LIN {X 0,Y 573.244,Z 41.075,A -85,B 0,C 180,E1 -2290.525,E2 -2290.525} C_VEL
LIN {X 0,Y 573.235,Z 41.08,A -85,B 0,C 180,E1 -2293.359,E2 -2293.359} C_VEL
LIN {X 0,Y 573.243,Z 41.074,A -85,B 0,C 180,E1 -2296.331,E2 -2296.331} C_VEL
LIN {X 0,Y 573.273,Z 41.079,A -85,B 0,C 180,E1 -2299.477,E2 -2299.477} C_VEL
LIN {X 0,Y 573.234,Z 41.075,A -85,B 0,C 180,E1 -2302.192,E2 -2302.192} C_VEL
LIN {X 0,Y 573.268,Z 41.075,A -85,B 0,C 180,E1 -2304.816,E2 -2304.816} C_VEL
LIN {X 0,Y 573.253,Z 41.079,A -85,B 0,C 180,E1 -2307.355,E2 -2307.355} C_VEL
LIN {X 0,Y 573.245,Z 41.076,A -85,B 0,C 180,E1 -2310.511,E2 -2310.511} C_VEL
LIN {X 0,Y 573.249,Z 41.08,A -85,B 0,C 180,E1 -2313.024,E2 -2313.024} C_VEL
LIN {X 0,Y 573.273,Z 41.072,A -85,B 0,C 180,E1 -2315.366,E2 -2315.366} C_VEL
LIN {X 0,Y 573.228,Z 41.081,A -85,B 0,C 180,E1 -2318.419,E2 -2318.419} C_VEL
LIN {X 0,Y 573.276,Z 41.076,A -85,B 0,C 180,E1 -2320.728,E2 -2320.728} C_VEL
LIN {X 0,Y 573.25,Z 41.073,A -85,B 0,C 180,E1 -2323.622,E2 -2323.622} C_VEL
LIN {X 0,Y 573.271,Z 41.073,A -85,B 0,C 180,E1 -2325.807,E2 -2325.807} C_VEL
LIN {X 0,Y 573.261,Z 41.074,A -85,B 0,C 180,E1 -2328.745,E2 -2328.745} C_VEL
LIN {X 0,Y 573.288,Z 41.07,A -85,B 0,C 180,E1 -2331.541,E2 -2331.541} C_VEL
LIN {X 0,Y 573.285,Z 41.073,A -85,B 0,C 180,E1 -2334.372,E2 -2334.372} C_VEL
LIN {X 0,Y 573.305,Z 41.075,A -85,B 0,C 180,E1 -2337.893,E2 -2337.893} C_VEL
LIN {X 0,Y 573.327,Z 41.064,A -85,B 0,C 180,E1 -2340.703,E2 -2340.703} C_VEL
LIN {X 0,Y 573.233,Z 41.082,A -85,B 0,C 180,E1 -2343.515,E2 -2343.515} C_VEL
LIN {X 0,Y 573.285,Z 41.076,A -85,B 0,C 180,E1 -2345.628,E2 -2345.628} C_VEL
LIN {X 0,Y 573.264,Z 41.075,A -85,B 0,C 180,E1 -2347.75,E2 -2347.75} C_VEL
LIN {X 0,Y 573.262,Z 41.073,A -85,B 0,C 180,E1 -2350.597,E2 -2350.597} C_VEL
LIN {X 0,Y 573.261,Z 41.074,A -85,B 0,C 180,E1 -2352.749,E2 -2352.749} C_VEL
LIN {X 0,Y 573.233,Z 41.082,A -85,B 0,C 180,E1 -2354.92,E2 -2354.92} C_VEL
LIN {X 0,Y 573.237,Z 41.074,A -85,B 0,C 180,E1 -2357.849,E2 -2357.849} C_VEL
LIN {X 0,Y 573.24,Z 41.075,A -85,B 0,C 180,E1 -2360.077,E2 -2360.077} C_VEL
LIN {X 0,Y 573.23,Z 41.078,A -85,B 0,C 180,E1 -2362.338,E2 -2362.338} C_VEL
LIN {X 0,Y 573.244,Z 41.079,A -85,B 0,C 180,E1 -2364.382,E2 -2364.382} C_VEL
LIN {X 0,Y 572.614,Z 41.163,A -85,B 0,C 180,E1 -2364.968,E2 -2364.968} C_VEL
LIN {X 0,Y 569.754,Z 41.518,A -85,B 0,C 180,E1 -2365.919,E2 -2365.919} C_VEL
LIN {X 0,Y 567.309,Z 41.822,A -85,B 0,C 180,E1 -2366.685,E2 -2366.685} C_VEL
LIN {X 0,Y 566.253,Z 41.947,A -85,B 0,C 180,E1 -2367.276,E2 -2367.276} C_VEL
LIN {X 0,Y 566.165,Z 41.956,A -85,B 0,C 180,E1 -2367.476,E2 -2367.476} C_VEL
LIN {X 0,Y 566.198,Z 41.952,A -85,B 0,C 180,E1 -2369.769,E2 -2369.769} C_VEL
LIN {X 0,Y 566.202,Z 41.96,A -85,B 0,C 180,E1 -2372.43,E2 -2372.43} C_VEL
LIN {X 0,Y 566.168,Z 41.956,A -85,B 0,C 180,E1 -2374.988,E2 -2374.988} C_VEL
LIN {X 0,Y 566.191,Z 41.954,A -85,B 0,C 180,E1 -2377.462,E2 -2377.462} C_VEL
LIN {X 0,Y 566.206,Z 41.957,A -85,B 0,C 180,E1 -2380.2,E2 -2380.2} C_VEL
LIN {X 0,Y 566.178,Z 41.956,A -85,B 0,C 180,E1 -2383.057,E2 -2383.057} C_VEL
LIN {X 0,Y 566.159,Z 41.964,A -85,B 0,C 180,E1 -2386.054,E2 -2386.054} C_VEL
LIN {X 0,Y 566.158,Z 41.958,A -85,B 0,C 180,E1 -2388.859,E2 -2388.859} C_VEL
LIN {X 0,Y 566.201,Z 41.96,A -85,B 0,C 180,E1 -2391.444,E2 -2391.444} C_VEL
LIN {X 0,Y 566.144,Z 41.96,A -85,B 0,C 180,E1 -2394.307,E2 -2394.307} C_VEL
LIN {X 0,Y 566.194,Z 41.958,A -85,B 0,C 180,E1 -2396.896,E2 -2396.896} C_VEL
LIN {X 0,Y 566.213,Z 42.062,A -85,B 0,C 180,E1 -2398.293,E2 -2398.293} C_VEL
LIN {X 0,Y 566.339,Z 48.784,A -85,B 0,C 180,E1 -2399.623,E2 -2399.623} C_VEL
LIN {X 0,Y 566.243,Z 61.213,A -85,B 0,C 180,E1 -2402.061,E2 -2402.061} C_VEL
LIN {X 0,Y 567.205,Z 67.215,A -85,B 0,C 180,E1 -2402.163,E2 -2402.163} C_VEL
LIN {X 0,Y 566.982,Z 167.233,A -85,B 0,C 180,E1 -2403.452,E2 -2403.452} C_VEL
LIN {X 0,Y 566.828,Z 180.305,A -85,B 0,C 180,E1 -2403.763,E2 -2403.763} C_VEL
LIN {X 0,Y 566.757,Z 193.318,A -85,B 0,C 180,E1 -2404.229,E2 -2404.229} C_VEL
LIN {X 0,Y 566.573,Z 205.2,A -85,B 0,C 180,E1 -2404.81,E2 -2404.81} C_VEL
LIN {X 0,Y 566.359,Z 216.706,A -85,B 0,C 180,E1 -2405.534,E2 -2405.534} C_VEL
LIN {X 0,Y 566.298,Z 227.724,A -85,B 0,C 180,E1 -2406.407,E2 -2406.407} C_VEL
LIN {X 0,Y 566.15,Z 237.413,A -85,B 0,C 180,E1 -2407.368,E2 -2407.368} C_VEL
LIN {X 0,Y 566.067,Z 245.994,A -85,B 0,C 180,E1 -2408.416,E2 -2408.416} C_VEL
LIN {X 0,Y 566.006,Z 252.944,A -85,B 0,C 180,E1 -2409.466,E2 -2409.466} C_VEL
LIN {X 0,Y 565.942,Z 259.355,A -85,B 0,C 180,E1 -2410.699,E2 -2410.699} C_VEL
LIN {X 0,Y 565.913,Z 264.167,A -85,B 0,C 180,E1 -2411.913,E2 -2411.913} C_VEL
LIN {X 0,Y 565.862,Z 267.344,A -85,B 0,C 180,E1 -2413.008,E2 -2413.008} C_VEL
LIN {X 0,Y 565.813,Z 269.563,A -85,B 0,C 180,E1 -2414.142,E2 -2414.142} C_VEL
LIN {X 0,Y 565.807,Z 270.469,A -85,B 0,C 180,E1 -2414.88,E2 -2414.88} C_VEL
LIN {X 0,Y 565.855,Z 270.917,A -85,B 0,C 180,E1 -2415.645,E2 -2415.645} C_VEL
LIN {X 0,Y 565.866,Z 270.938,A -85,B 0,C 180,E1 -2416.351,E2 -2416.351} C_VEL
LIN {X 0,Y 565.845,Z 270.566,A -85,B 0,C 180,E1 -2417.082,E2 -2417.082} C_VEL
LIN {X 0,Y 565.867,Z 269.774,A -85,B 0,C 180,E1 -2417.811,E2 -2417.811} C_VEL
LIN {X 0,Y 565.908,Z 267.91,A -85,B 0,C 180,E1 -2418.845,E2 -2418.845} C_VEL
LIN {X 0,Y 565.925,Z 264.812,A -85,B 0,C 180,E1 -2419.988,E2 -2419.988} C_VEL
LIN {X 0,Y 565.944,Z 260.793,A -85,B 0,C 180,E1 -2421.07,E2 -2421.07} C_VEL
LIN {X 0,Y 565.986,Z 254.613,A -85,B 0,C 180,E1 -2422.329,E2 -2422.329} C_VEL
LIN {X 0,Y 566.023,Z 248.098,A -85,B 0,C 180,E1 -2423.377,E2 -2423.377} C_VEL
LIN {X 0,Y 566.099,Z 239.606,A -85,B 0,C 180,E1 -2424.479,E2 -2424.479} C_VEL
LIN {X 0,Y 566.237,Z 231.088,A -85,B 0,C 180,E1 -2425.373,E2 -2425.373} C_VEL
LIN {X 0,Y 566.385,Z 220.63,A -85,B 0,C 180,E1 -2426.265,E2 -2426.265} C_VEL
LIN {X 0,Y 566.535,Z 210.305,A -85,B 0,C 180,E1 -2426.978,E2 -2426.978} C_VEL
LIN {X 0,Y 566.7,Z 199.046,A -85,B 0,C 180,E1 -2427.601,E2 -2427.601} C_VEL
LIN {X 0,Y 566.746,Z 187.532,A -85,B 0,C 180,E1 -2428.09,E2 -2428.09} C_VEL
LIN {X 0,Y 566.884,Z 175.12,A -85,B 0,C 180,E1 -2428.468,E2 -2428.468} C_VEL
LIN {X 0,Y 566.961,Z 162.555,A -85,B 0,C 180,E1 -2428.713,E2 -2428.713} C_VEL
LIN {X 0,Y 567.066,Z 66.094,A -85,B 0,C 180,E1 -2429.945,E2 -2429.945} C_VEL
LIN {X 0,Y 566.19,Z 61.097,A -85,B 0,C 180,E1 -2430.045,E2 -2430.045} C_VEL
LIN {X 0,Y 566.414,Z 46.902,A -85,B 0,C 180,E1 -2432.845,E2 -2432.845} C_VEL
LIN {X 0,Y 566.211,Z 41.956,A -85,B 0,C 180,E1 -2433.826,E2 -2433.826} C_VEL
LIN {X 0,Y 566.26,Z 41.946,A -85,B 0,C 180,E1 -2435.699,E2 -2435.699} C_VEL
LIN {X 0,Y 566.232,Z 41.957,A -85,B 0,C 180,E1 -2438.566,E2 -2438.566} C_VEL
LIN {X 0,Y 566.249,Z 41.945,A -85,B 0,C 180,E1 -2441.454,E2 -2441.454} C_VEL
LIN {X 0,Y 566.241,Z 41.955,A -85,B 0,C 180,E1 -2444.506,E2 -2444.506} C_VEL
LIN {X 0,Y 566.204,Z 41.951,A -85,B 0,C 180,E1 -2447.332,E2 -2447.332} C_VEL
LIN {X 0,Y 566.212,Z 41.958,A -85,B 0,C 180,E1 -2450.337,E2 -2450.337} C_VEL
LIN {X 0,Y 566.175,Z 41.955,A -85,B 0,C 180,E1 -2453.281,E2 -2453.281} C_VEL
LIN {X 0,Y 566.215,Z 41.954,A -85,B 0,C 180,E1 -2455.749,E2 -2455.749} C_VEL
LIN {X 0,Y 566.209,Z 41.956,A -85,B 0,C 180,E1 -2458.202,E2 -2458.202} C_VEL
LIN {X 0,Y 566.195,Z 41.952,A -85,B 0,C 180,E1 -2461.076,E2 -2461.076} C_VEL
LIN {X 0,Y 566.218,Z 41.958,A -85,B 0,C 180,E1 -2463.734,E2 -2463.734} C_VEL
LIN {X 0,Y 566.212,Z 41.95,A -85,B 0,C 180,E1 -2466.569,E2 -2466.569} C_VEL
LIN {X 0,Y 566.218,Z 41.957,A -85,B 0,C 180,E1 -2469.685,E2 -2469.685} C_VEL
LIN {X 0,Y 566.205,Z 41.953,A -85,B 0,C 180,E1 -2472.917,E2 -2472.917} C_VEL
LIN {X 0,Y 566.198,Z 41.952,A -85,B 0,C 180,E1 -2476.049,E2 -2476.049} C_VEL
LIN {X 0,Y 566.207,Z 41.96,A -85,B 0,C 180,E1 -2479.214,E2 -2479.214} C_VEL
LIN {X 0,Y 566.19,Z 41.955,A -85,B 0,C 180,E1 -2481.637,E2 -2481.637} C_VEL
LIN {X 0,Y 566.167,Z 41.956,A -85,B 0,C 180,E1 -2484.308,E2 -2484.308} C_VEL
LIN {X 0,Y 566.223,Z 41.957,A -85,B 0,C 180,E1 -2486.898,E2 -2486.898} C_VEL
LIN {X 0,Y 566.184,Z 41.955,A -85,B 0,C 180,E1 -2489.407,E2 -2489.407} C_VEL
LIN {X 0,Y 566.215,Z 41.949,A -85,B 0,C 180,E1 -2491.857,E2 -2491.857} C_VEL
LIN {X 0,Y 566.213,Z 41.953,A -85,B 0,C 180,E1 -2494.251,E2 -2494.251} C_VEL
LIN {X 0,Y 566.176,Z 41.962,A -85,B 0,C 180,E1 -2496.718,E2 -2496.718} C_VEL
LIN {X 0,Y 566.215,Z 41.95,A -85,B 0,C 180,E1 -2499.663,E2 -2499.663} C_VEL
LIN {X 0,Y 566.201,Z 41.956,A -85,B 0,C 180,E1 -2502.668,E2 -2502.668} C_VEL
LIN {X 0,Y 566.237,Z 41.948,A -85,B 0,C 180,E1 -2505.627,E2 -2505.627} C_VEL
LIN {X 0,Y 566.238,Z 41.949,A -85,B 0,C 180,E1 -2508.675,E2 -2508.675} C_VEL
LIN {X 0,Y 566.23,Z 41.949,A -85,B 0,C 180,E1 -2511.434,E2 -2511.434} C_VEL
LIN {X 0,Y 566.256,Z 41.949,A -85,B 0,C 180,E1 -2514.301,E2 -2514.301} C_VEL
LIN {X 0,Y 566.28,Z 41.951,A -85,B 0,C 180,E1 -2517.866,E2 -2517.866} C_VEL
LIN {X 0,Y 566.301,Z 41.939,A -85,B 0,C 180,E1 -2520.711,E2 -2520.711} C_VEL
LIN {X 0,Y 566.27,Z 41.943,A -85,B 0,C 180,E1 -2522.845,E2 -2522.845} C_VEL
LIN {X 0,Y 566.255,Z 41.952,A -85,B 0,C 180,E1 -2525.698,E2 -2525.698} C_VEL
LIN {X 0,Y 566.207,Z 41.95,A -85,B 0,C 180,E1 -2528.566,E2 -2528.566} C_VEL
LIN {X 0,Y 566.244,Z 41.954,A -85,B 0,C 180,E1 -2531.454,E2 -2531.454} C_VEL
LIN {X 0,Y 566.232,Z 41.948,A -85,B 0,C 180,E1 -2534.505,E2 -2534.505} C_VEL
LIN {X 0,Y 566.2,Z 41.958,A -85,B 0,C 180,E1 -2537.332,E2 -2537.332} C_VEL
LIN {X 0,Y 566.209,Z 41.951,A -85,B 0,C 180,E1 -2540.337,E2 -2540.337} C_VEL
LIN {X 0,Y 566.17,Z 41.96,A -85,B 0,C 180,E1 -2543.281,E2 -2543.281} C_VEL
LIN {X 0,Y 566.208,Z 41.95,A -85,B 0,C 180,E1 -2545.749,E2 -2545.749} C_VEL
LIN {X 0,Y 566.205,Z 41.952,A -85,B 0,C 180,E1 -2548.202,E2 -2548.202} C_VEL
LIN {X 0,Y 566.192,Z 41.956,A -85,B 0,C 180,E1 -2551.076,E2 -2551.076} C_VEL
LIN {X 0,Y 566.213,Z 41.95,A -85,B 0,C 180,E1 -2553.734,E2 -2553.734} C_VEL
LIN {X 0,Y 566.202,Z 41.96,A -85,B 0,C 180,E1 -2556.57,E2 -2556.57} C_VEL
LIN {X 0,Y 566.217,Z 41.95,A -85,B 0,C 180,E1 -2559.686,E2 -2559.686} C_VEL
LIN {X 0,Y 566.203,Z 41.952,A -85,B 0,C 180,E1 -2562.917,E2 -2562.917} C_VEL
LIN {X 0,Y 566.196,Z 41.96,A -85,B 0,C 180,E1 -2566.049,E2 -2566.049} C_VEL
LIN {X 0,Y 566.206,Z 41.951,A -85,B 0,C 180,E1 -2569.215,E2 -2569.215} C_VEL
LIN {X 0,Y 566.184,Z 41.958,A -85,B 0,C 180,E1 -2571.636,E2 -2571.636} C_VEL
LIN {X 0,Y 566.165,Z 41.959,A -85,B 0,C 180,E1 -2574.308,E2 -2574.308} C_VEL
LIN {X 0,Y 566.208,Z 41.95,A -85,B 0,C 180,E1 -2576.897,E2 -2576.897} C_VEL
LIN {X 0,Y 566.177,Z 41.959,A -85,B 0,C 180,E1 -2579.407,E2 -2579.407} C_VEL
LIN {X 0,Y 566.215,Z 41.957,A -85,B 0,C 180,E1 -2581.857,E2 -2581.857} C_VEL
LIN {X 0,Y 566.21,Z 41.954,A -85,B 0,C 180,E1 -2584.251,E2 -2584.251} C_VEL
LIN {X 0,Y 566.261,Z 42.133,A -85,B 0,C 180,E1 -2585.676,E2 -2585.676} C_VEL
LIN {X 0,Y 567.069,Z 47.897,A -85,B 0,C 180,E1 -2586.509,E2 -2586.509} C_VEL
LIN {X 0,Y 566.843,Z 66.898,A -85,B 0,C 180,E1 -2589.117,E2 -2589.117} C_VEL
LIN {X 0,Y 566.688,Z 87.811,A -85,B 0,C 180,E1 -2591.938,E2 -2591.938} C_VEL
LIN {X 0,Y 566.434,Z 110.038,A -85,B 0,C 180,E1 -2594.897,E2 -2594.897} C_VEL
LIN {X 0,Y 566.431,Z 118.271,A -85,B 0,C 180,E1 -2595.987,E2 -2595.987} C_VEL
LIN {X 0,Y 567.159,Z 125.154,A -85,B 0,C 180,E1 -2596.095,E2 -2596.095} C_VEL
LIN {X 0,Y 566.941,Z 226.934,A -85,B 0,C 180,E1 -2597.402,E2 -2597.402} C_VEL
LIN {X 0,Y 566.859,Z 240.209,A -85,B 0,C 180,E1 -2597.719,E2 -2597.719} C_VEL
LIN {X 0,Y 566.76,Z 252.371,A -85,B 0,C 180,E1 -2598.148,E2 -2598.148} C_VEL
LIN {X 0,Y 566.604,Z 264.234,A -85,B 0,C 180,E1 -2598.712,E2 -2598.712} C_VEL
LIN {X 0,Y 566.442,Z 276.19,A -85,B 0,C 180,E1 -2599.455,E2 -2599.455} C_VEL
LIN {X 0,Y 566.325,Z 286.603,A -85,B 0,C 180,E1 -2600.265,E2 -2600.265} C_VEL
LIN {X 0,Y 566.207,Z 295.111,A -85,B 0,C 180,E1 -2601.074,E2 -2601.074} C_VEL
LIN {X 0,Y 566.112,Z 302.959,A -85,B 0,C 180,E1 -2601.971,E2 -2601.971} C_VEL
LIN {X 0,Y 566.004,Z 310.621,A -85,B 0,C 180,E1 -2603.046,E2 -2603.046} C_VEL
LIN {X 0,Y 566.004,Z 317.678,A -85,B 0,C 180,E1 -2604.299,E2 -2604.299} C_VEL
LIN {X 0,Y 565.933,Z 322.372,A -85,B 0,C 180,E1 -2605.37,E2 -2605.37} C_VEL
LIN {X 0,Y 565.927,Z 325.958,A -85,B 0,C 180,E1 -2606.44,E2 -2606.44} C_VEL
LIN {X 0,Y 565.878,Z 327.807,A -85,B 0,C 180,E1 -2607.152,E2 -2607.152} C_VEL
LIN {X 0,Y 565.846,Z 330.183,A -85,B 0,C 180,E1 -2608.576,E2 -2608.576} C_VEL
LIN {X 0,Y 565.839,Z 331,A -85,B 0,C 180,E1 -2610,E2 -2610} C_VEL
LIN {X 0,Y 565.846,Z 330.185,A -85,B 0,C 180,E1 -2611.423,E2 -2611.423} C_VEL
LIN {X 0,Y 565.878,Z 327.811,A -85,B 0,C 180,E1 -2612.847,E2 -2612.847} C_VEL
LIN {X 0,Y 565.926,Z 324.896,A -85,B 0,C 180,E1 -2613.916,E2 -2613.916} C_VEL
LIN {X 0,Y 565.878,Z 320.949,A -85,B 0,C 180,E1 -2614.987,E2 -2614.987} C_VEL
LIN {X 0,Y 566.004,Z 315.869,A -85,B 0,C 180,E1 -2616.058,E2 -2616.058} C_VEL
LIN {X 0,Y 566.04,Z 309.469,A -85,B 0,C 180,E1 -2617.132,E2 -2617.132} C_VEL
LIN {X 0,Y 566.133,Z 301.48,A -85,B 0,C 180,E1 -2618.207,E2 -2618.207} C_VEL
LIN {X 0,Y 566.228,Z 293.336,A -85,B 0,C 180,E1 -2619.105,E2 -2619.105} C_VEL
LIN {X 0,Y 566.342,Z 283.401,A -85,B 0,C 180,E1 -2620.005,E2 -2620.005} C_VEL
LIN {X 0,Y 566.514,Z 272.293,A -85,B 0,C 180,E1 -2620.807,E2 -2620.807} C_VEL
LIN {X 0,Y 566.612,Z 261.177,A -85,B 0,C 180,E1 -2621.446,E2 -2621.446} C_VEL
LIN {X 0,Y 566.738,Z 248.984,A -85,B 0,C 180,E1 -2621.988,E2 -2621.988} C_VEL
LIN {X 0,Y 566.886,Z 236.185,A -85,B 0,C 180,E1 -2622.394,E2 -2622.394} C_VEL
LIN {X 0,Y 566.99,Z 224.122,A -85,B 0,C 180,E1 -2622.641,E2 -2622.641} C_VEL
LIN {X 0,Y 567.069,Z 122.874,A -85,B 0,C 180,E1 -2623.937,E2 -2623.937} C_VEL
LIN {X 0,Y 566.429,Z 118.184,A -85,B 0,C 180,E1 -2624.024,E2 -2624.024} C_VEL
LIN {X 0,Y 566.582,Z 96.456,A -85,B 0,C 180,E1 -2626.903,E2 -2626.903} C_VEL
LIN {X 0,Y 566.79,Z 75.205,A -85,B 0,C 180,E1 -2629.748,E2 -2629.748} C_VEL
LIN {X 0,Y 566.963,Z 54.272,A -85,B 0,C 180,E1 -2632.598,E2 -2632.598} C_VEL
LIN {X 0,Y 566.957,Z 45.828,A -85,B 0,C 180,E1 -2633.766,E2 -2633.766} C_VEL
LIN {X 0,Y 566.256,Z 41.954,A -85,B 0,C 180,E1 -2634.348,E2 -2634.348} C_VEL
LIN {X 0,Y 566.213,Z 41.952,A -85,B 0,C 180,E1 -2637.339,E2 -2637.339} C_VEL
LIN {X 0,Y 566.201,Z 41.955,A -85,B 0,C 180,E1 -2639.768,E2 -2639.768} C_VEL
LIN {X 0,Y 566.204,Z 41.957,A -85,B 0,C 180,E1 -2642.429,E2 -2642.429} C_VEL
LIN {X 0,Y 566.212,Z 41.95,A -85,B 0,C 180,E1 -2644.994,E2 -2644.994} C_VEL
LIN {X 0,Y 566.197,Z 41.955,A -85,B 0,C 180,E1 -2647.46,E2 -2647.46} C_VEL
LIN {X 0,Y 566.206,Z 41.955,A -85,B 0,C 180,E1 -2650.199,E2 -2650.199} C_VEL
LIN {X 0,Y 566.199,Z 41.953,A -85,B 0,C 180,E1 -2653.054,E2 -2653.054} C_VEL
LIN {X 0,Y 566.197,Z 41.954,A -85,B 0,C 180,E1 -2656.048,E2 -2656.048} C_VEL
LIN {X 0,Y 566.207,Z 41.952,A -85,B 0,C 180,E1 -2658.863,E2 -2658.863} C_VEL
LIN {X 0,Y 566.188,Z 41.957,A -85,B 0,C 180,E1 -2661.637,E2 -2661.637} C_VEL
LIN {X 0,Y 566.212,Z 41.95,A -85,B 0,C 180,E1 -2664.311,E2 -2664.311} C_VEL
LIN {X 0,Y 566.227,Z 41.954,A -85,B 0,C 180,E1 -2666.898,E2 -2666.898} C_VEL
LIN {X 0,Y 566.183,Z 41.957,A -85,B 0,C 180,E1 -2669.407,E2 -2669.407} C_VEL
LIN {X 0,Y 566.227,Z 41.948,A -85,B 0,C 180,E1 -2671.858,E2 -2671.858} C_VEL
LIN {X 0,Y 566.212,Z 41.951,A -85,B 0,C 180,E1 -2674.251,E2 -2674.251} C_VEL
LIN {X 0,Y 566.189,Z 41.961,A -85,B 0,C 180,E1 -2676.714,E2 -2676.714} C_VEL
LIN {X 0,Y 566.212,Z 41.95,A -85,B 0,C 180,E1 -2679.663,E2 -2679.663} C_VEL
LIN {X 0,Y 566.198,Z 41.958,A -85,B 0,C 180,E1 -2682.668,E2 -2682.668} C_VEL
LIN {X 0,Y 566.232,Z 41.948,A -85,B 0,C 180,E1 -2685.627,E2 -2685.627} C_VEL
LIN {X 0,Y 566.233,Z 41.95,A -85,B 0,C 180,E1 -2688.675,E2 -2688.675} C_VEL
LIN {X 0,Y 566.232,Z 41.948,A -85,B 0,C 180,E1 -2691.434,E2 -2691.434} C_VEL
LIN {X 0,Y 566.254,Z 41.95,A -85,B 0,C 180,E1 -2694.302,E2 -2694.302} C_VEL
LIN {X 0,Y 566.276,Z 41.95,A -85,B 0,C 180,E1 -2697.866,E2 -2697.866} C_VEL
LIN {X 0,Y 566.298,Z 41.939,A -85,B 0,C 180,E1 -2700.711,E2 -2700.711} C_VEL
LIN {X 0,Y 566.268,Z 41.942,A -85,B 0,C 180,E1 -2702.846,E2 -2702.846} C_VEL
LIN {X 0,Y 566.252,Z 41.951,A -85,B 0,C 180,E1 -2705.699,E2 -2705.699} C_VEL
LIN {X 0,Y 566.199,Z 41.951,A -85,B 0,C 180,E1 -2708.566,E2 -2708.566} C_VEL
LIN {X 0,Y 566.24,Z 41.952,A -85,B 0,C 180,E1 -2711.455,E2 -2711.455} C_VEL
LIN {X 0,Y 566.227,Z 41.949,A -85,B 0,C 180,E1 -2714.505,E2 -2714.505} C_VEL
LIN {X 0,Y 566.196,Z 41.956,A -85,B 0,C 180,E1 -2717.332,E2 -2717.332} C_VEL
LIN {X 0,Y 566.206,Z 41.953,A -85,B 0,C 180,E1 -2720.338,E2 -2720.338} C_VEL
LIN {X 0,Y 566.167,Z 41.958,A -85,B 0,C 180,E1 -2723.281,E2 -2723.281} C_VEL
LIN {X 0,Y 566.203,Z 41.95,A -85,B 0,C 180,E1 -2725.75,E2 -2725.75} C_VEL
LIN {X 0,Y 566.165,Z 41.956,A -85,B 0,C 180,E1 -2727.476,E2 -2727.476} C_VEL
LIN {X 0,Y 565.495,Z 42.044,A -85,B 0,C 180,E1 -2728.07,E2 -2728.07} C_VEL
LIN {X 0,Y 562.644,Z 42.396,A -85,B 0,C 180,E1 -2729.034,E2 -2729.034} C_VEL
LIN {X 0,Y 560.242,Z 42.696,A -85,B 0,C 180,E1 -2729.81,E2 -2729.81} C_VEL
LIN {X 0,Y 559.217,Z 42.83,A -85,B 0,C 180,E1 -2730.409,E2 -2730.409} C_VEL
LIN {X 0,Y 559.136,Z 42.833,A -85,B 0,C 180,E1 -2730.612,E2 -2730.612} C_VEL
LIN {X 0,Y 559.152,Z 42.834,A -85,B 0,C 180,E1 -2732.716,E2 -2732.716} C_VEL
LIN {X 0,Y 559.117,Z 42.833,A -85,B 0,C 180,E1 -2735.325,E2 -2735.325} C_VEL
LIN {X 0,Y 559.129,Z 42.841,A -85,B 0,C 180,E1 -2738.018,E2 -2738.018} C_VEL
LIN {X 0,Y 559.152,Z 42.829,A -85,B 0,C 180,E1 -2740.813,E2 -2740.813} C_VEL
LIN {X 0,Y 559.107,Z 42.844,A -85,B 0,C 180,E1 -2743.738,E2 -2743.738} C_VEL
LIN {X 0,Y 559.111,Z 42.839,A -85,B 0,C 180,E1 -2746.264,E2 -2746.264} C_VEL
LIN {X 0,Y 559.143,Z 42.832,A -85,B 0,C 180,E1 -2748.952,E2 -2748.952} C_VEL
LIN {X 0,Y 559.169,Z 42.832,A -85,B 0,C 180,E1 -2751.193,E2 -2751.193} C_VEL
LIN {X 0,Y 559.118,Z 42.84,A -85,B 0,C 180,E1 -2753.788,E2 -2753.788} C_VEL
LIN {X 0,Y 559.146,Z 42.834,A -85,B 0,C 180,E1 -2756.424,E2 -2756.424} C_VEL
LIN {X 0,Y 559.189,Z 42.862,A -85,B 0,C 180,E1 -2758.177,E2 -2758.177} C_VEL
LIN {X 0,Y 559.371,Z 49.056,A -85,B 0,C 180,E1 -2759.413,E2 -2759.413} C_VEL
LIN {X 0,Y 559.253,Z 61.716,A -85,B 0,C 180,E1 -2761.884,E2 -2761.884} C_VEL
LIN {X 0,Y 560.318,Z 68.245,A -85,B 0,C 180,E1 -2761.997,E2 -2761.997} C_VEL
LIN {X 0,Y 560.067,Z 167.692,A -85,B 0,C 180,E1 -2763.296,E2 -2763.296} C_VEL
LIN {X 0,Y 559.917,Z 180.86,A -85,B 0,C 180,E1 -2763.615,E2 -2763.615} C_VEL
LIN {X 0,Y 559.82,Z 193.819,A -85,B 0,C 180,E1 -2764.085,E2 -2764.085} C_VEL
LIN {X 0,Y 559.637,Z 204.826,A -85,B 0,C 180,E1 -2764.625,E2 -2764.625} C_VEL
LIN {X 0,Y 559.42,Z 215.758,A -85,B 0,C 180,E1 -2765.31,E2 -2765.31} C_VEL
LIN {X 0,Y 559.315,Z 226.96,A -85,B 0,C 180,E1 -2766.193,E2 -2766.193} C_VEL
LIN {X 0,Y 559.161,Z 235.94,A -85,B 0,C 180,E1 -2767.069,E2 -2767.069} C_VEL
LIN {X 0,Y 559.031,Z 245.321,A -85,B 0,C 180,E1 -2768.209,E2 -2768.209} C_VEL
LIN {X 0,Y 558.926,Z 253.046,A -85,B 0,C 180,E1 -2769.386,E2 -2769.386} C_VEL
LIN {X 0,Y 558.877,Z 259.176,A -85,B 0,C 180,E1 -2770.587,E2 -2770.587} C_VEL
LIN {X 0,Y 558.815,Z 263.53,A -85,B 0,C 180,E1 -2771.675,E2 -2771.675} C_VEL
LIN {X 0,Y 558.772,Z 267.225,A -85,B 0,C 180,E1 -2772.922,E2 -2772.922} C_VEL
LIN {X 0,Y 558.731,Z 269.278,A -85,B 0,C 180,E1 -2773.935,E2 -2773.935} C_VEL
LIN {X 0,Y 558.711,Z 270.272,A -85,B 0,C 180,E1 -2774.683,E2 -2774.683} C_VEL
LIN {X 0,Y 558.762,Z 270.904,A -85,B 0,C 180,E1 -2775.581,E2 -2775.581} C_VEL
LIN {X 0,Y 558.745,Z 270.686,A -85,B 0,C 180,E1 -2776.915,E2 -2776.915} C_VEL
LIN {X 0,Y 558.773,Z 269.995,A -85,B 0,C 180,E1 -2777.654,E2 -2777.654} C_VEL
LIN {X 0,Y 558.806,Z 268.044,A -85,B 0,C 180,E1 -2778.813,E2 -2778.813} C_VEL
LIN {X 0,Y 558.847,Z 264.18,A -85,B 0,C 180,E1 -2780.226,E2 -2780.226} C_VEL
LIN {X 0,Y 558.86,Z 259.98,A -85,B 0,C 180,E1 -2781.321,E2 -2781.321} C_VEL
LIN {X 0,Y 558.928,Z 253.647,A -85,B 0,C 180,E1 -2782.595,E2 -2782.595} C_VEL
LIN {X 0,Y 559.026,Z 246.759,A -85,B 0,C 180,E1 -2783.685,E2 -2783.685} C_VEL
LIN {X 0,Y 559.115,Z 238.158,A -85,B 0,C 180,E1 -2784.772,E2 -2784.772} C_VEL
LIN {X 0,Y 559.219,Z 229.38,A -85,B 0,C 180,E1 -2785.676,E2 -2785.676} C_VEL
LIN {X 0,Y 559.405,Z 219.736,A -85,B 0,C 180,E1 -2786.489,E2 -2786.489} C_VEL
LIN {X 0,Y 559.587,Z 209.178,A -85,B 0,C 180,E1 -2787.211,E2 -2787.211} C_VEL
LIN {X 0,Y 559.751,Z 197.391,A -85,B 0,C 180,E1 -2787.842,E2 -2787.842} C_VEL
LIN {X 0,Y 559.857,Z 185.182,A -85,B 0,C 180,E1 -2788.337,E2 -2788.337} C_VEL
LIN {X 0,Y 559.988,Z 172.547,A -85,B 0,C 180,E1 -2788.697,E2 -2788.697} C_VEL
LIN {X 0,Y 560.101,Z 159.151,A -85,B 0,C 180,E1 -2788.922,E2 -2788.922} C_VEL
LIN {X 0,Y 560.186,Z 66.943,A -85,B 0,C 180,E1 -2790.113,E2 -2790.113} C_VEL
LIN {X 0,Y 559.196,Z 61.451,A -85,B 0,C 180,E1 -2790.225,E2 -2790.225} C_VEL
LIN {X 0,Y 559.422,Z 46.188,A -85,B 0,C 180,E1 -2793.241,E2 -2793.241} C_VEL
LIN {X 0,Y 559.174,Z 42.833,A -85,B 0,C 180,E1 -2793.919,E2 -2793.919} C_VEL
LIN {X 0,Y 559.23,Z 42.822,A -85,B 0,C 180,E1 -2795.77,E2 -2795.77} C_VEL
LIN {X 0,Y 559.191,Z 42.834,A -85,B 0,C 180,E1 -2798.675,E2 -2798.675} C_VEL
LIN {X 0,Y 559.212,Z 42.822,A -85,B 0,C 180,E1 -2801.601,E2 -2801.601} C_VEL
LIN {X 0,Y 559.207,Z 42.829,A -85,B 0,C 180,E1 -2804.596,E2 -2804.596} C_VEL
LIN {X 0,Y 559.147,Z 42.83,A -85,B 0,C 180,E1 -2807.558,E2 -2807.558} C_VEL
LIN {X 0,Y 559.172,Z 42.83,A -85,B 0,C 180,E1 -2809.838,E2 -2809.838} C_VEL
LIN {X 0,Y 559.147,Z 42.839,A -85,B 0,C 180,E1 -2812.153,E2 -2812.153} C_VEL
LIN {X 0,Y 559.181,Z 42.826,A -85,B 0,C 180,E1 -2815.298,E2 -2815.298} C_VEL
LIN {X 0,Y 559.187,Z 42.83,A -85,B 0,C 180,E1 -2817.712,E2 -2817.712} C_VEL
LIN {X 0,Y 559.158,Z 42.834,A -85,B 0,C 180,E1 -2820.183,E2 -2820.183} C_VEL
LIN {X 0,Y 559.161,Z 42.828,A -85,B 0,C 180,E1 -2822.715,E2 -2822.715} C_VEL
LIN {X 0,Y 559.15,Z 42.833,A -85,B 0,C 180,E1 -2825.323,E2 -2825.323} C_VEL
LIN {X 0,Y 559.135,Z 42.835,A -85,B 0,C 180,E1 -2828.018,E2 -2828.018} C_VEL
LIN {X 0,Y 559.16,Z 42.829,A -85,B 0,C 180,E1 -2830.812,E2 -2830.812} C_VEL
LIN {X 0,Y 559.142,Z 42.835,A -85,B 0,C 180,E1 -2833.734,E2 -2833.734} C_VEL
LIN {X 0,Y 559.149,Z 42.832,A -85,B 0,C 180,E1 -2836.803,E2 -2836.803} C_VEL
LIN {X 0,Y 559.159,Z 42.838,A -85,B 0,C 180,E1 -2839.187,E2 -2839.187} C_VEL
LIN {X 0,Y 559.137,Z 42.831,A -85,B 0,C 180,E1 -2841.982,E2 -2841.982} C_VEL
LIN {X 0,Y 559.136,Z 42.837,A -85,B 0,C 180,E1 -2844.787,E2 -2844.787} C_VEL
LIN {X 0,Y 559.159,Z 42.832,A -85,B 0,C 180,E1 -2847.364,E2 -2847.364} C_VEL
LIN {X 0,Y 559.152,Z 42.83,A -85,B 0,C 180,E1 -2850.142,E2 -2850.142} C_VEL
LIN {X 0,Y 559.172,Z 42.831,A -85,B 0,C 180,E1 -2853.097,E2 -2853.097} C_VEL
LIN {X 0,Y 559.16,Z 42.828,A -85,B 0,C 180,E1 -2855.495,E2 -2855.495} C_VEL
LIN {X 0,Y 559.176,Z 42.835,A -85,B 0,C 180,E1 -2858.624,E2 -2858.624} C_VEL
LIN {X 0,Y 559.165,Z 42.83,A -85,B 0,C 180,E1 -2860.926,E2 -2860.926} C_VEL
LIN {X 0,Y 559.167,Z 42.831,A -85,B 0,C 180,E1 -2863.948,E2 -2863.948} C_VEL
LIN {X 0,Y 559.173,Z 42.835,A -85,B 0,C 180,E1 -2866.184,E2 -2866.184} C_VEL
LIN {X 0,Y 559.199,Z 42.824,A -85,B 0,C 180,E1 -2869.133,E2 -2869.133} C_VEL
LIN {X 0,Y 559.202,Z 42.833,A -85,B 0,C 180,E1 -2872.053,E2 -2872.053} C_VEL
LIN {X 0,Y 559.253,Z 42.817,A -85,B 0,C 180,E1 -2874.953,E2 -2874.953} C_VEL
LIN {X 0,Y 559.251,Z 42.826,A -85,B 0,C 180,E1 -2877.839,E2 -2877.839} C_VEL
LIN {X 0,Y 559.272,Z 42.814,A -85,B 0,C 180,E1 -2880.72,E2 -2880.72} C_VEL
LIN {X 0,Y 559.237,Z 42.819,A -85,B 0,C 180,E1 -2882.881,E2 -2882.881} C_VEL
LIN {X 0,Y 559.224,Z 42.827,A -85,B 0,C 180,E1 -2885.77,E2 -2885.77} C_VEL
LIN {X 0,Y 559.172,Z 42.827,A -85,B 0,C 180,E1 -2888.675,E2 -2888.675} C_VEL
LIN {X 0,Y 559.208,Z 42.828,A -85,B 0,C 180,E1 -2891.6,E2 -2891.6} C_VEL
LIN {X 0,Y 559.203,Z 42.824,A -85,B 0,C 180,E1 -2894.595,E2 -2894.595} C_VEL
LIN {X 0,Y 559.143,Z 42.834,A -85,B 0,C 180,E1 -2897.557,E2 -2897.557} C_VEL
LIN {X 0,Y 559.168,Z 42.828,A -85,B 0,C 180,E1 -2899.837,E2 -2899.837} C_VEL
LIN {X 0,Y 559.142,Z 42.831,A -85,B 0,C 180,E1 -2902.153,E2 -2902.153} C_VEL
LIN {X 0,Y 559.177,Z 42.83,A -85,B 0,C 180,E1 -2905.298,E2 -2905.298} C_VEL
LIN {X 0,Y 559.17,Z 42.83,A -85,B 0,C 180,E1 -2908.381,E2 -2908.381} C_VEL
LIN {X 0,Y 559.147,Z 42.832,A -85,B 0,C 180,E1 -2911.273,E2 -2911.273} C_VEL
LIN {X 0,Y 559.167,Z 42.829,A -85,B 0,C 180,E1 -2913.949,E2 -2913.949} C_VEL
LIN {X 0,Y 559.142,Z 42.832,A -85,B 0,C 180,E1 -2917.108,E2 -2917.108} C_VEL
LIN {X 0,Y 559.162,Z 42.831,A -85,B 0,C 180,E1 -2919.942,E2 -2919.942} C_VEL
LIN {X 0,Y 559.159,Z 42.831,A -85,B 0,C 180,E1 -2922.744,E2 -2922.744} C_VEL
LIN {X 0,Y 559.149,Z 42.833,A -85,B 0,C 180,E1 -2925.761,E2 -2925.761} C_VEL
LIN {X 0,Y 559.164,Z 42.835,A -85,B 0,C 180,E1 -2928.23,E2 -2928.23} C_VEL
LIN {X 0,Y 559.174,Z 42.827,A -85,B 0,C 180,E1 -2931.192,E2 -2931.192} C_VEL
LIN {X 0,Y 559.141,Z 42.838,A -85,B 0,C 180,E1 -2933.789,E2 -2933.789} C_VEL
LIN {X 0,Y 559.161,Z 42.83,A -85,B 0,C 180,E1 -2936.425,E2 -2936.425} C_VEL
LIN {X 0,Y 559.155,Z 42.83,A -85,B 0,C 180,E1 -2938.98,E2 -2938.98} C_VEL
LIN {X 0,Y 559.171,Z 42.838,A -85,B 0,C 180,E1 -2941.619,E2 -2941.619} C_VEL
LIN {X 0,Y 559.18,Z 42.833,A -85,B 0,C 180,E1 -2943.903,E2 -2943.903} C_VEL
LIN {X 0,Y 559.209,Z 42.84,A -85,B 0,C 180,E1 -2945.497,E2 -2945.497} C_VEL
LIN {X 0,Y 560.118,Z 48.575,A -85,B 0,C 180,E1 -2946.342,E2 -2946.342} C_VEL
LIN {X 0,Y 559.88,Z 66.551,A -85,B 0,C 180,E1 -2948.845,E2 -2948.845} C_VEL
LIN {X 0,Y 559.699,Z 86.063,A -85,B 0,C 180,E1 -2951.515,E2 -2951.515} C_VEL
LIN {X 0,Y 559.486,Z 106.914,A -85,B 0,C 180,E1 -2954.331,E2 -2954.331} C_VEL
LIN {X 0,Y 559.374,Z 117.904,A -85,B 0,C 180,E1 -2955.806,E2 -2955.806} C_VEL
LIN {X 0,Y 560.269,Z 125.801,A -85,B 0,C 180,E1 -2955.934,E2 -2955.934} C_VEL
LIN {X 0,Y 560.033,Z 226.62,A -85,B 0,C 180,E1 -2957.244,E2 -2957.244} C_VEL
LIN {X 0,Y 559.922,Z 239.939,A -85,B 0,C 180,E1 -2957.564,E2 -2957.564} C_VEL
LIN {X 0,Y 559.812,Z 252.152,A -85,B 0,C 180,E1 -2957.999,E2 -2957.999} C_VEL
LIN {X 0,Y 559.622,Z 263.89,A -85,B 0,C 180,E1 -2958.559,E2 -2958.559} C_VEL
LIN {X 0,Y 559.456,Z 276.101,A -85,B 0,C 180,E1 -2959.322,E2 -2959.322} C_VEL
LIN {X 0,Y 559.305,Z 286.586,A -85,B 0,C 180,E1 -2960.142,E2 -2960.142} C_VEL
LIN {X 0,Y 559.162,Z 295.111,A -85,B 0,C 180,E1 -2960.961,E2 -2960.961} C_VEL
LIN {X 0,Y 559.05,Z 302.959,A -85,B 0,C 180,E1 -2961.869,E2 -2961.869} C_VEL
LIN {X 0,Y 558.944,Z 310.621,A -85,B 0,C 180,E1 -2962.958,E2 -2962.958} C_VEL
LIN {X 0,Y 558.936,Z 317.678,A -85,B 0,C 180,E1 -2964.227,E2 -2964.227} C_VEL
LIN {X 0,Y 558.826,Z 322.372,A -85,B 0,C 180,E1 -2965.311,E2 -2965.311} C_VEL
LIN {X 0,Y 558.836,Z 325.957,A -85,B 0,C 180,E1 -2966.395,E2 -2966.395} C_VEL
LIN {X 0,Y 558.799,Z 327.806,A -85,B 0,C 180,E1 -2967.116,E2 -2967.116} C_VEL
LIN {X 0,Y 558.745,Z 330.182,A -85,B 0,C 180,E1 -2968.558,E2 -2968.558} C_VEL
LIN {X 0,Y 558.74,Z 331,A -85,B 0,C 180,E1 -2970,E2 -2970} C_VEL
LIN {X 0,Y 558.745,Z 330.184,A -85,B 0,C 180,E1 -2971.441,E2 -2971.441} C_VEL
LIN {X 0,Y 558.799,Z 327.811,A -85,B 0,C 180,E1 -2972.883,E2 -2972.883} C_VEL
LIN {X 0,Y 558.844,Z 324.896,A -85,B 0,C 180,E1 -2973.966,E2 -2973.966} C_VEL
LIN {X 0,Y 558.798,Z 320.949,A -85,B 0,C 180,E1 -2975.051,E2 -2975.051} C_VEL
LIN {X 0,Y 558.923,Z 315.869,A -85,B 0,C 180,E1 -2976.135,E2 -2976.135} C_VEL
LIN {X 0,Y 558.977,Z 309.468,A -85,B 0,C 180,E1 -2977.223,E2 -2977.223} C_VEL
LIN {X 0,Y 559.098,Z 301.479,A -85,B 0,C 180,E1 -2978.311,E2 -2978.311} C_VEL
LIN {X 0,Y 559.194,Z 293.335,A -85,B 0,C 180,E1 -2979.221,E2 -2979.221} C_VEL
LIN {X 0,Y 559.353,Z 283.362,A -85,B 0,C 180,E1 -2980.131,E2 -2980.131} C_VEL
LIN {X 0,Y 559.524,Z 272.286,A -85,B 0,C 180,E1 -2980.937,E2 -2980.937} C_VEL
LIN {X 0,Y 559.671,Z 260.275,A -85,B 0,C 180,E1 -2981.627,E2 -2981.627} C_VEL
LIN {X 0,Y 559.808,Z 247.523,A -85,B 0,C 180,E1 -2982.185,E2 -2982.185} C_VEL
LIN {X 0,Y 559.999,Z 234.053,A -85,B 0,C 180,E1 -2982.595,E2 -2982.595} C_VEL
LIN {X 0,Y 560.105,Z 220.755,A -85,B 0,C 180,E1 -2982.846,E2 -2982.846} C_VEL
LIN {X 0,Y 560.211,Z 123.819,A -85,B 0,C 180,E1 -2984.093,E2 -2984.093} C_VEL
LIN {X 0,Y 559.352,Z 117.793,A -85,B 0,C 180,E1 -2984.205,E2 -2984.205} C_VEL
LIN {X 0,Y 559.578,Z 96.415,A -85,B 0,C 180,E1 -2987.075,E2 -2987.075} C_VEL
LIN {X 0,Y 559.834,Z 74.819,A -85,B 0,C 180,E1 -2990.004,E2 -2990.004} C_VEL
LIN {X 0,Y 560.077,Z 52.515,A -85,B 0,C 180,E1 -2993.087,E2 -2993.087} C_VEL
LIN {X 0,Y 559.952,Z 46.915,A -85,B 0,C 180,E1 -2993.876,E2 -2993.876} C_VEL
LIN {X 0,Y 559.206,Z 42.832,A -85,B 0,C 180,E1 -2994.502,E2 -2994.502} C_VEL
LIN {X 0,Y 559.17,Z 42.832,A -85,B 0,C 180,E1 -2996.902,E2 -2996.902} C_VEL
LIN {X 0,Y 559.149,Z 42.835,A -85,B 0,C 180,E1 -2999.857,E2 -2999.857} C_VEL
LIN {X 0,Y 559.153,Z 42.832,A -85,B 0,C 180,E1 -3002.715,E2 -3002.715} C_VEL
LIN {X 0,Y 559.157,Z 42.83,A -85,B 0,C 180,E1 -3005.322,E2 -3005.322} C_VEL
LIN {X 0,Y 559.133,Z 42.84,A -85,B 0,C 180,E1 -3008.017,E2 -3008.017} C_VEL
LIN {X 0,Y 559.155,Z 42.83,A -85,B 0,C 180,E1 -3010.812,E2 -3010.812} C_VEL
LIN {X 0,Y 559.155,Z 42.837,A -85,B 0,C 180,E1 -3013.732,E2 -3013.732} C_VEL
LIN {X 0,Y 559.145,Z 42.83,A -85,B 0,C 180,E1 -3016.803,E2 -3016.803} C_VEL
LIN {X 0,Y 559.174,Z 42.832,A -85,B 0,C 180,E1 -3019.189,E2 -3019.189} C_VEL
LIN {X 0,Y 559.133,Z 42.832,A -85,B 0,C 180,E1 -3021.982,E2 -3021.982} C_VEL
LIN {X 0,Y 559.159,Z 42.832,A -85,B 0,C 180,E1 -3024.783,E2 -3024.783} C_VEL
LIN {X 0,Y 559.172,Z 42.833,A -85,B 0,C 180,E1 -3027.361,E2 -3027.361} C_VEL
LIN {X 0,Y 559.147,Z 42.83,A -85,B 0,C 180,E1 -3030.142,E2 -3030.142} C_VEL
LIN {X 0,Y 559.168,Z 42.833,A -85,B 0,C 180,E1 -3033.098,E2 -3033.098} C_VEL
LIN {X 0,Y 559.155,Z 42.83,A -85,B 0,C 180,E1 -3035.495,E2 -3035.495} C_VEL
LIN {X 0,Y 559.17,Z 42.835,A -85,B 0,C 180,E1 -3038.624,E2 -3038.624} C_VEL
LIN {X 0,Y 559.166,Z 42.83,A -85,B 0,C 180,E1 -3040.926,E2 -3040.926} C_VEL
LIN {X 0,Y 559.165,Z 42.83,A -85,B 0,C 180,E1 -3043.948,E2 -3043.948} C_VEL
LIN {X 0,Y 559.17,Z 42.835,A -85,B 0,C 180,E1 -3046.184,E2 -3046.184} C_VEL
LIN {X 0,Y 559.195,Z 42.824,A -85,B 0,C 180,E1 -3049.134,E2 -3049.134} C_VEL
LIN {X 0,Y 559.2,Z 42.831,A -85,B 0,C 180,E1 -3052.054,E2 -3052.054} C_VEL
LIN {X 0,Y 559.251,Z 42.817,A -85,B 0,C 180,E1 -3054.953,E2 -3054.953} C_VEL
LIN {X 0,Y 559.248,Z 42.825,A -85,B 0,C 180,E1 -3057.84,E2 -3057.84} C_VEL
LIN {X 0,Y 559.269,Z 42.815,A -85,B 0,C 180,E1 -3060.72,E2 -3060.72} C_VEL
LIN {X 0,Y 559.235,Z 42.818,A -85,B 0,C 180,E1 -3062.882,E2 -3062.882} C_VEL
LIN {X 0,Y 559.221,Z 42.826,A -85,B 0,C 180,E1 -3065.77,E2 -3065.77} C_VEL
LIN {X 0,Y 559.164,Z 42.827,A -85,B 0,C 180,E1 -3068.675,E2 -3068.675} C_VEL
LIN {X 0,Y 559.204,Z 42.826,A -85,B 0,C 180,E1 -3071.601,E2 -3071.601} C_VEL
LIN {X 0,Y 559.199,Z 42.826,A -85,B 0,C 180,E1 -3074.596,E2 -3074.596} C_VEL
LIN {X 0,Y 559.139,Z 42.832,A -85,B 0,C 180,E1 -3077.558,E2 -3077.558} C_VEL
LIN {X 0,Y 559.164,Z 42.828,A -85,B 0,C 180,E1 -3079.838,E2 -3079.838} C_VEL
LIN {X 0,Y 559.138,Z 42.831,A -85,B 0,C 180,E1 -3082.153,E2 -3082.153} C_VEL
LIN {X 0,Y 559.173,Z 42.827,A -85,B 0,C 180,E1 -3085.299,E2 -3085.299} C_VEL
LIN {X 0,Y 559.126,Z 42.833,A -85,B 0,C 180,E1 -3087.716,E2 -3087.716} C_VEL
LIN {X 0,Y 559.136,Z 42.833,A -85,B 0,C 180,E1 -3090.612,E2 -3090.612} C_VEL
LIN {X 0,Y 558.474,Z 42.917,A -85,B 0,C 180,E1 -3091.213,E2 -3091.213} C_VEL
LIN {X 0,Y 555.609,Z 43.278,A -85,B 0,C 180,E1 -3092.189,E2 -3092.189} C_VEL
LIN {X 0,Y 553.194,Z 43.574,A -85,B 0,C 180,E1 -3092.975,E2 -3092.975} C_VEL
LIN {X 0,Y 552.173,Z 43.7,A -85,B 0,C 180,E1 -3093.582,E2 -3093.582} C_VEL
LIN {X 0,Y 552.099,Z 43.711,A -85,B 0,C 180,E1 -3093.787,E2 -3093.787} C_VEL
LIN {X 0,Y 552.097,Z 43.711,A -85,B 0,C 180,E1 -3096.748,E2 -3096.748} C_VEL
LIN {X 0,Y 552.127,Z 43.708,A -85,B 0,C 180,E1 -3099.528,E2 -3099.528} C_VEL
LIN {X 0,Y 552.107,Z 43.712,A -85,B 0,C 180,E1 -3102.428,E2 -3102.428} C_VEL
LIN {X 0,Y 552.075,Z 43.716,A -85,B 0,C 180,E1 -3105.561,E2 -3105.561} C_VEL
LIN {X 0,Y 552.078,Z 43.712,A -85,B 0,C 180,E1 -3108.551,E2 -3108.551} C_VEL
LIN {X 0,Y 552.111,Z 43.715,A -85,B 0,C 180,E1 -3111.411,E2 -3111.411} C_VEL
LIN {X 0,Y 552.072,Z 43.715,A -85,B 0,C 180,E1 -3114.156,E2 -3114.156} C_VEL
LIN {X 0,Y 552.105,Z 43.713,A -85,B 0,C 180,E1 -3116.814,E2 -3116.814} C_VEL
LIN {X 0,Y 552.144,Z 43.822,A -85,B 0,C 180,E1 -3118.086,E2 -3118.086} C_VEL
LIN {X 0,Y 552.416,Z 48.267,A -85,B 0,C 180,E1 -3118.986,E2 -3118.986} C_VEL
LIN {X 0,Y 552.245,Z 61.901,A -85,B 0,C 180,E1 -3121.698,E2 -3121.698} C_VEL
LIN {X 0,Y 553.449,Z 69.602,A -85,B 0,C 180,E1 -3121.832,E2 -3121.832} C_VEL
LIN {X 0,Y 553.156,Z 168.314,A -85,B 0,C 180,E1 -3123.139,E2 -3123.139} C_VEL
LIN {X 0,Y 553.022,Z 181.84,A -85,B 0,C 180,E1 -3123.476,E2 -3123.476} C_VEL
LIN {X 0,Y 552.882,Z 194.315,A -85,B 0,C 180,E1 -3123.938,E2 -3123.938} C_VEL
LIN {X 0,Y 552.674,Z 206.196,A -85,B 0,C 180,E1 -3124.538,E2 -3124.538} C_VEL
LIN {X 0,Y 552.45,Z 217.596,A -85,B 0,C 180,E1 -3125.278,E2 -3125.278} C_VEL
LIN {X 0,Y 552.34,Z 227.73,A -85,B 0,C 180,E1 -3126.101,E2 -3126.101} C_VEL
LIN {X 0,Y 552.157,Z 236.371,A -85,B 0,C 180,E1 -3126.959,E2 -3126.959} C_VEL
LIN {X 0,Y 552.036,Z 244.482,A -85,B 0,C 180,E1 -3127.941,E2 -3127.941} C_VEL
LIN {X 0,Y 551.882,Z 252.298,A -85,B 0,C 180,E1 -3129.111,E2 -3129.111} C_VEL
LIN {X 0,Y 551.839,Z 258.229,A -85,B 0,C 180,E1 -3130.225,E2 -3130.225} C_VEL
LIN {X 0,Y 551.737,Z 263.254,A -85,B 0,C 180,E1 -3131.431,E2 -3131.431} C_VEL
LIN {X 0,Y 551.689,Z 267.419,A -85,B 0,C 180,E1 -3132.831,E2 -3132.831} C_VEL
LIN {X 0,Y 551.671,Z 269.289,A -85,B 0,C 180,E1 -3133.724,E2 -3133.724} C_VEL
LIN {X 0,Y 551.631,Z 270.356,A -85,B 0,C 180,E1 -3134.482,E2 -3134.482} C_VEL
LIN {X 0,Y 551.677,Z 271.163,A -85,B 0,C 180,E1 -3135.512,E2 -3135.512} C_VEL
LIN {X 0,Y 551.658,Z 271.08,A -85,B 0,C 180,E1 -3136.744,E2 -3136.744} C_VEL
LIN {X 0,Y 551.682,Z 270.474,A -85,B 0,C 180,E1 -3137.493,E2 -3137.493} C_VEL
LIN {X 0,Y 551.722,Z 268.497,A -85,B 0,C 180,E1 -3138.772,E2 -3138.772} C_VEL
LIN {X 0,Y 551.771,Z 265.117,A -85,B 0,C 180,E1 -3140.099,E2 -3140.099} C_VEL
LIN {X 0,Y 551.779,Z 261.134,A -85,B 0,C 180,E1 -3141.209,E2 -3141.209} C_VEL
LIN {X 0,Y 551.876,Z 254.996,A -85,B 0,C 180,E1 -3142.5,E2 -3142.5} C_VEL
LIN {X 0,Y 551.953,Z 248.599,A -85,B 0,C 180,E1 -3143.564,E2 -3143.564} C_VEL
LIN {X 0,Y 552.074,Z 240.087,A -85,B 0,C 180,E1 -3144.705,E2 -3144.705} C_VEL
LIN {X 0,Y 552.213,Z 231.616,A -85,B 0,C 180,E1 -3145.621,E2 -3145.621} C_VEL
LIN {X 0,Y 552.43,Z 221.191,A -85,B 0,C 180,E1 -3146.536,E2 -3146.536} C_VEL
LIN {X 0,Y 552.639,Z 210.875,A -85,B 0,C 180,E1 -3147.267,E2 -3147.267} C_VEL
LIN {X 0,Y 552.829,Z 199.561,A -85,B 0,C 180,E1 -3147.906,E2 -3147.906} C_VEL
LIN {X 0,Y 552.924,Z 187.937,A -85,B 0,C 180,E1 -3148.407,E2 -3148.407} C_VEL
LIN {X 0,Y 553.07,Z 175.398,A -85,B 0,C 180,E1 -3148.794,E2 -3148.794} C_VEL
LIN {X 0,Y 553.163,Z 162.531,A -85,B 0,C 180,E1 -3149.045,E2 -3149.045} C_VEL
LIN {X 0,Y 553.327,Z 67.776,A -85,B 0,C 180,E1 -3150.285,E2 -3150.285} C_VEL
LIN {X 0,Y 552.205,Z 61.789,A -85,B 0,C 180,E1 -3150.41,E2 -3150.41} C_VEL
LIN {X 0,Y 552.422,Z 47.323,A -85,B 0,C 180,E1 -3153.282,E2 -3153.282} C_VEL
LIN {X 0,Y 552.136,Z 43.71,A -85,B 0,C 180,E1 -3154.015,E2 -3154.015} C_VEL
LIN {X 0,Y 552.201,Z 43.698,A -85,B 0,C 180,E1 -3155.844,E2 -3155.844} C_VEL
LIN {X 0,Y 552.158,Z 43.708,A -85,B 0,C 180,E1 -3158.786,E2 -3158.786} C_VEL
LIN {X 0,Y 552.169,Z 43.7,A -85,B 0,C 180,E1 -3161.751,E2 -3161.751} C_VEL
LIN {X 0,Y 552.143,Z 43.707,A -85,B 0,C 180,E1 -3164.748,E2 -3164.748} C_VEL
LIN {X 0,Y 552.105,Z 43.709,A -85,B 0,C 180,E1 -3167.789,E2 -3167.789} C_VEL
LIN {X 0,Y 552.132,Z 43.711,A -85,B 0,C 180,E1 -3170.101,E2 -3170.101} C_VEL
LIN {X 0,Y 552.098,Z 43.713,A -85,B 0,C 180,E1 -3172.451,E2 -3172.451} C_VEL
LIN {X 0,Y 552.161,Z 43.701,A -85,B 0,C 180,E1 -3175.35,E2 -3175.35} C_VEL
LIN {X 0,Y 552.113,Z 43.714,A -85,B 0,C 180,E1 -3178.098,E2 -3178.098} C_VEL
LIN {X 0,Y 552.107,Z 43.708,A -85,B 0,C 180,E1 -3180.609,E2 -3180.609} C_VEL
LIN {X 0,Y 552.121,Z 43.707,A -85,B 0,C 180,E1 -3183.186,E2 -3183.186} C_VEL
LIN {X 0,Y 552.105,Z 43.714,A -85,B 0,C 180,E1 -3185.842,E2 -3185.842} C_VEL
LIN {X 0,Y 552.125,Z 43.707,A -85,B 0,C 180,E1 -3189.061,E2 -3189.061} C_VEL
LIN {X 0,Y 552.125,Z 43.714,A -85,B 0,C 180,E1 -3191.446,E2 -3191.446} C_VEL
LIN {X 0,Y 552.093,Z 43.709,A -85,B 0,C 180,E1 -3194.531,E2 -3194.531} C_VEL
LIN {X 0,Y 552.134,Z 43.708,A -85,B 0,C 180,E1 -3197.584,E2 -3197.584} C_VEL
LIN {X 0,Y 552.137,Z 43.704,A -85,B 0,C 180,E1 -3200.473,E2 -3200.473} C_VEL
LIN {X 0,Y 552.11,Z 43.712,A -85,B 0,C 180,E1 -3203.317,E2 -3203.317} C_VEL
LIN {X 0,Y 552.131,Z 43.704,A -85,B 0,C 180,E1 -3205.939,E2 -3205.939} C_VEL
LIN {X 0,Y 552.123,Z 43.709,A -85,B 0,C 180,E1 -3208.54,E2 -3208.54} C_VEL
LIN {X 0,Y 552.128,Z 43.706,A -85,B 0,C 180,E1 -3211.438,E2 -3211.438} C_VEL
LIN {X 0,Y 552.132,Z 43.708,A -85,B 0,C 180,E1 -3214.356,E2 -3214.356} C_VEL
LIN {X 0,Y 552.107,Z 43.714,A -85,B 0,C 180,E1 -3216.758,E2 -3216.758} C_VEL
LIN {X 0,Y 552.123,Z 43.706,A -85,B 0,C 180,E1 -3219.12,E2 -3219.12} C_VEL
LIN {X 0,Y 552.123,Z 43.705,A -85,B 0,C 180,E1 -3221.444,E2 -3221.444} C_VEL
LIN {X 0,Y 552.118,Z 43.707,A -85,B 0,C 180,E1 -3223.737,E2 -3223.737} C_VEL
LIN {X 0,Y 552.138,Z 43.708,A -85,B 0,C 180,E1 -3226.004,E2 -3226.004} C_VEL
LIN {X 0,Y 552.166,Z 43.7,A -85,B 0,C 180,E1 -3228.993,E2 -3228.993} C_VEL
LIN {X 0,Y 552.157,Z 43.708,A -85,B 0,C 180,E1 -3231.951,E2 -3231.951} C_VEL
LIN {X 0,Y 552.228,Z 43.692,A -85,B 0,C 180,E1 -3234.889,E2 -3234.889} C_VEL
LIN {X 0,Y 552.223,Z 43.701,A -85,B 0,C 180,E1 -3237.812,E2 -3237.812} C_VEL
LIN {X 0,Y 552.242,Z 43.69,A -85,B 0,C 180,E1 -3240.729,E2 -3240.729} C_VEL
LIN {X 0,Y 552.204,Z 43.695,A -85,B 0,C 180,E1 -3242.918,E2 -3242.918} C_VEL
LIN {X 0,Y 552.195,Z 43.701,A -85,B 0,C 180,E1 -3245.844,E2 -3245.844} C_VEL
LIN {X 0,Y 552.147,Z 43.703,A -85,B 0,C 180,E1 -3248.786,E2 -3248.786} C_VEL
LIN {X 0,Y 552.165,Z 43.704,A -85,B 0,C 180,E1 -3251.75,E2 -3251.75} C_VEL
LIN {X 0,Y 552.139,Z 43.705,A -85,B 0,C 180,E1 -3254.748,E2 -3254.748} C_VEL
LIN {X 0,Y 552.101,Z 43.709,A -85,B 0,C 180,E1 -3257.789,E2 -3257.789} C_VEL
LIN {X 0,Y 552.129,Z 43.704,A -85,B 0,C 180,E1 -3260.101,E2 -3260.101} C_VEL
LIN {X 0,Y 552.093,Z 43.711,A -85,B 0,C 180,E1 -3262.451,E2 -3262.451} C_VEL
LIN {X 0,Y 552.139,Z 43.706,A -85,B 0,C 180,E1 -3265.346,E2 -3265.346} C_VEL
LIN {X 0,Y 552.1,Z 43.709,A -85,B 0,C 180,E1 -3268.099,E2 -3268.099} C_VEL
LIN {X 0,Y 552.104,Z 43.715,A -85,B 0,C 180,E1 -3270.609,E2 -3270.609} C_VEL
LIN {X 0,Y 552.114,Z 43.708,A -85,B 0,C 180,E1 -3273.186,E2 -3273.186} C_VEL
LIN {X 0,Y 552.088,Z 43.71,A -85,B 0,C 180,E1 -3275.844,E2 -3275.844} C_VEL
LIN {X 0,Y 552.119,Z 43.712,A -85,B 0,C 180,E1 -3278.589,E2 -3278.589} C_VEL
LIN {X 0,Y 552.122,Z 43.705,A -85,B 0,C 180,E1 -3281.446,E2 -3281.446} C_VEL
LIN {X 0,Y 552.09,Z 43.714,A -85,B 0,C 180,E1 -3284.531,E2 -3284.531} C_VEL
LIN {X 0,Y 552.132,Z 43.706,A -85,B 0,C 180,E1 -3287.585,E2 -3287.585} C_VEL
LIN {X 0,Y 552.13,Z 43.707,A -85,B 0,C 180,E1 -3290.473,E2 -3290.473} C_VEL
LIN {X 0,Y 552.109,Z 43.708,A -85,B 0,C 180,E1 -3293.317,E2 -3293.317} C_VEL
LIN {X 0,Y 552.129,Z 43.712,A -85,B 0,C 180,E1 -3295.939,E2 -3295.939} C_VEL
LIN {X 0,Y 552.122,Z 43.705,A -85,B 0,C 180,E1 -3298.541,E2 -3298.541} C_VEL
LIN {X 0,Y 552.127,Z 43.713,A -85,B 0,C 180,E1 -3301.438,E2 -3301.438} C_VEL
LIN {X 0,Y 552.131,Z 43.708,A -85,B 0,C 180,E1 -3304.356,E2 -3304.356} C_VEL
LIN {X 0,Y 552.234,Z 43.895,A -85,B 0,C 180,E1 -3305.368,E2 -3305.368} C_VEL
LIN {X 0,Y 553.186,Z 50.087,A -85,B 0,C 180,E1 -3306.292,E2 -3306.292} C_VEL
LIN {X 0,Y 552.927,Z 69.004,A -85,B 0,C 180,E1 -3308.957,E2 -3308.957} C_VEL
LIN {X 0,Y 552.652,Z 91.274,A -85,B 0,C 180,E1 -3312.038,E2 -3312.038} C_VEL
LIN {X 0,Y 552.365,Z 112.348,A -85,B 0,C 180,E1 -3314.918,E2 -3314.918} C_VEL
LIN {X 0,Y 552.327,Z 117.508,A -85,B 0,C 180,E1 -3315.62,E2 -3315.62} C_VEL
LIN {X 0,Y 553.384,Z 125.621,A -85,B 0,C 180,E1 -3315.758,E2 -3315.758} C_VEL
LIN {X 0,Y 553.119,Z 226.206,A -85,B 0,C 180,E1 -3317.082,E2 -3317.082} C_VEL
LIN {X 0,Y 552.973,Z 239.536,A -85,B 0,C 180,E1 -3317.405,E2 -3317.405} C_VEL
LIN {X 0,Y 552.849,Z 251.746,A -85,B 0,C 180,E1 -3317.845,E2 -3317.845} C_VEL
LIN {X 0,Y 552.649,Z 262.668,A -85,B 0,C 180,E1 -3318.368,E2 -3318.368} C_VEL
LIN {X 0,Y 552.45,Z 274.41,A -85,B 0,C 180,E1 -3319.092,E2 -3319.092} C_VEL
LIN {X 0,Y 552.258,Z 285.12,A -85,B 0,C 180,E1 -3319.922,E2 -3319.922} C_VEL
LIN {X 0,Y 552.11,Z 294.774,A -85,B 0,C 180,E1 -3320.844,E2 -3320.844} C_VEL
LIN {X 0,Y 551.984,Z 302.692,A -85,B 0,C 180,E1 -3321.765,E2 -3321.765} C_VEL
LIN {X 0,Y 551.889,Z 310.427,A -85,B 0,C 180,E1 -3322.867,E2 -3322.867} C_VEL
LIN {X 0,Y 551.845,Z 317.561,A -85,B 0,C 180,E1 -3324.152,E2 -3324.152} C_VEL
LIN {X 0,Y 551.723,Z 322.302,A -85,B 0,C 180,E1 -3325.25,E2 -3325.25} C_VEL
LIN {X 0,Y 551.75,Z 325.931,A -85,B 0,C 180,E1 -3326.348,E2 -3326.348} C_VEL
LIN {X 0,Y 551.723,Z 327.795,A -85,B 0,C 180,E1 -3327.079,E2 -3327.079} C_VEL
LIN {X 0,Y 551.645,Z 330.179,A -85,B 0,C 180,E1 -3328.54,E2 -3328.54} C_VEL
LIN {X 0,Y 551.64,Z 331,A -85,B 0,C 180,E1 -3330,E2 -3330} C_VEL
LIN {X 0,Y 551.645,Z 330.182,A -85,B 0,C 180,E1 -3331.46,E2 -3331.46} C_VEL
LIN {X 0,Y 551.723,Z 327.799,A -85,B 0,C 180,E1 -3332.92,E2 -3332.92} C_VEL
LIN {X 0,Y 551.764,Z 324.859,A -85,B 0,C 180,E1 -3334.017,E2 -3334.017} C_VEL
LIN {X 0,Y 551.723,Z 320.862,A -85,B 0,C 180,E1 -3335.115,E2 -3335.115} C_VEL
LIN {X 0,Y 551.797,Z 315.034,A -85,B 0,C 180,E1 -3336.342,E2 -3336.342} C_VEL
LIN {X 0,Y 551.891,Z 308.015,A -85,B 0,C 180,E1 -3337.5,E2 -3337.5} C_VEL
LIN {X 0,Y 552.038,Z 299.694,A -85,B 0,C 180,E1 -3338.603,E2 -3338.603} C_VEL
LIN {X 0,Y 552.163,Z 291.166,A -85,B 0,C 180,E1 -3339.524,E2 -3339.524} C_VEL
LIN {X 0,Y 552.365,Z 280.635,A -85,B 0,C 180,E1 -3340.446,E2 -3340.446} C_VEL
LIN {X 0,Y 552.554,Z 268.64,A -85,B 0,C 180,E1 -3341.286,E2 -3341.286} C_VEL
LIN {X 0,Y 552.759,Z 256.878,A -85,B 0,C 180,E1 -3341.923,E2 -3341.923} C_VEL
LIN {X 0,Y 552.931,Z 244.495,A -85,B 0,C 180,E1 -3342.432,E2 -3342.432} C_VEL
LIN {X 0,Y 553.037,Z 231.791,A -85,B 0,C 180,E1 -3342.802,E2 -3342.802} C_VEL
LIN {X 0,Y 553.164,Z 218.524,A -85,B 0,C 180,E1 -3343.033,E2 -3343.033} C_VEL
LIN {X 0,Y 553.21,Z 123.836,A -85,B 0,C 180,E1 -3344.27,E2 -3344.27} C_VEL
LIN {X 0,Y 552.315,Z 117.342,A -85,B 0,C 180,E1 -3344.397,E2 -3344.397} C_VEL
LIN {X 0,Y 552.594,Z 94.763,A -85,B 0,C 180,E1 -3347.471,E2 -3347.471} C_VEL
LIN {X 0,Y 552.887,Z 74.46,A -85,B 0,C 180,E1 -3350.266,E2 -3350.266} C_VEL
LIN {X 0,Y 553.207,Z 51.199,A -85,B 0,C 180,E1 -3353.525,E2 -3353.525} C_VEL
LIN {X 0,Y 552.441,Z 45.114,A -85,B 0,C 180,E1 -3354.422,E2 -3354.422} C_VEL
LIN {X 0,Y 552.176,Z 43.708,A -85,B 0,C 180,E1 -3354.635,E2 -3354.635} C_VEL
LIN {X 0,Y 552.14,Z 43.705,A -85,B 0,C 180,E1 -3357.273,E2 -3357.273} C_VEL
LIN {X 0,Y 552.117,Z 43.714,A -85,B 0,C 180,E1 -3360.05,E2 -3360.05} C_VEL
LIN {X 0,Y 552.111,Z 43.709,A -85,B 0,C 180,E1 -3362.845,E2 -3362.845} C_VEL
LIN {X 0,Y 552.107,Z 43.709,A -85,B 0,C 180,E1 -3365.444,E2 -3365.444} C_VEL
LIN {X 0,Y 552.097,Z 43.717,A -85,B 0,C 180,E1 -3367.885,E2 -3367.885} C_VEL
LIN {X 0,Y 552.108,Z 43.709,A -85,B 0,C 180,E1 -3370.481,E2 -3370.481} C_VEL
LIN {X 0,Y 552.118,Z 43.712,A -85,B 0,C 180,E1 -3373.484,E2 -3373.484} C_VEL
LIN {X 0,Y 552.105,Z 43.706,A -85,B 0,C 180,E1 -3376.576,E2 -3376.576} C_VEL
LIN {X 0,Y 552.14,Z 43.711,A -85,B 0,C 180,E1 -3379.522,E2 -3379.522} C_VEL
LIN {X 0,Y 552.092,Z 43.708,A -85,B 0,C 180,E1 -3382.336,E2 -3382.336} C_VEL
LIN {X 0,Y 552.129,Z 43.712,A -85,B 0,C 180,E1 -3385.054,E2 -3385.054} C_VEL
LIN {X 0,Y 552.124,Z 43.707,A -85,B 0,C 180,E1 -3387.682,E2 -3387.682} C_VEL
LIN {X 0,Y 552.11,Z 43.707,A -85,B 0,C 180,E1 -3390.235,E2 -3390.235} C_VEL
LIN {X 0,Y 552.138,Z 43.71,A -85,B 0,C 180,E1 -3392.999,E2 -3392.999} C_VEL
LIN {X 0,Y 552.111,Z 43.711,A -85,B 0,C 180,E1 -3395.161,E2 -3395.161} C_VEL
LIN {X 0,Y 552.094,Z 43.707,A -85,B 0,C 180,E1 -3397.549,E2 -3397.549} C_VEL
LIN {X 0,Y 552.154,Z 43.708,A -85,B 0,C 180,E1 -3400.674,E2 -3400.674} C_VEL
LIN {X 0,Y 552.115,Z 43.707,A -85,B 0,C 180,E1 -3403.737,E2 -3403.737} C_VEL
LIN {X 0,Y 552.133,Z 43.708,A -85,B 0,C 180,E1 -3406.004,E2 -3406.004} C_VEL
LIN {X 0,Y 552.162,Z 43.701,A -85,B 0,C 180,E1 -3408.993,E2 -3408.993} C_VEL
LIN {X 0,Y 552.155,Z 43.708,A -85,B 0,C 180,E1 -3411.952,E2 -3411.952} C_VEL
LIN {X 0,Y 552.225,Z 43.693,A -85,B 0,C 180,E1 -3414.889,E2 -3414.889} C_VEL
LIN {X 0,Y 552.22,Z 43.7,A -85,B 0,C 180,E1 -3417.812,E2 -3417.812} C_VEL
LIN {X 0,Y 552.239,Z 43.691,A -85,B 0,C 180,E1 -3420.729,E2 -3420.729} C_VEL
LIN {X 0,Y 552.202,Z 43.694,A -85,B 0,C 180,E1 -3422.918,E2 -3422.918} C_VEL
LIN {X 0,Y 552.192,Z 43.701,A -85,B 0,C 180,E1 -3425.844,E2 -3425.844} C_VEL
LIN {X 0,Y 552.141,Z 43.703,A -85,B 0,C 180,E1 -3428.786,E2 -3428.786} C_VEL
LIN {X 0,Y 552.161,Z 43.702,A -85,B 0,C 180,E1 -3431.751,E2 -3431.751} C_VEL
LIN {X 0,Y 552.135,Z 43.707,A -85,B 0,C 180,E1 -3434.749,E2 -3434.749} C_VEL
LIN {X 0,Y 552.096,Z 43.708,A -85,B 0,C 180,E1 -3437.789,E2 -3437.789} C_VEL
LIN {X 0,Y 552.125,Z 43.706,A -85,B 0,C 180,E1 -3440.102,E2 -3440.102} C_VEL
LIN {X 0,Y 552.089,Z 43.712,A -85,B 0,C 180,E1 -3442.451,E2 -3442.451} C_VEL
LIN {X 0,Y 552.135,Z 43.703,A -85,B 0,C 180,E1 -3445.347,E2 -3445.347} C_VEL
LIN {X 0,Y 552.076,Z 43.714,A -85,B 0,C 180,E1 -3448.101,E2 -3448.101} C_VEL
LIN {X 0,Y 552.1,Z 43.715,A -85,B 0,C 180,E1 -3450.61,E2 -3450.61} C_VEL
LIN {X 0,Y 552.106,Z 43.708,A -85,B 0,C 180,E1 -3453.187,E2 -3453.187} C_VEL
LIN {X 0,Y 552.099,Z 43.711,A -85,B 0,C 180,E1 -3453.787,E2 -3453.787} C_VEL
LIN {X 0,Y 551.463,Z 43.795,A -85,B 0,C 180,E1 -3454.395,E2 -3454.395} C_VEL
LIN {X 0,Y 548.643,Z 44.146,A -85,B 0,C 180,E1 -3455.383,E2 -3455.383} C_VEL
LIN {X 0,Y 546.225,Z 44.448,A -85,B 0,C 180,E1 -3456.179,E2 -3456.179} C_VEL
LIN {X 0,Y 545.157,Z 44.575,A -85,B 0,C 180,E1 -3456.793,E2 -3456.793} C_VEL
LIN {X 0,Y 545.055,Z 44.587,A -85,B 0,C 180,E1 -3457,E2 -3457} C_VEL
LIN {X 0,Y 545.064,Z 44.591,A -85,B 0,C 180,E1 -3460.143,E2 -3460.143} C_VEL
LIN {X 0,Y 545.022,Z 44.592,A -85,B 0,C 180,E1 -3463.113,E2 -3463.113} C_VEL
LIN {X 0,Y 545.046,Z 44.592,A -85,B 0,C 180,E1 -3466.227,E2 -3466.227} C_VEL
LIN {X 0,Y 545.029,Z 44.59,A -85,B 0,C 180,E1 -3468.881,E2 -3468.881} C_VEL
LIN {X 0,Y 545.045,Z 44.595,A -85,B 0,C 180,E1 -3471.763,E2 -3471.763} C_VEL
LIN {X 0,Y 545.027,Z 44.592,A -85,B 0,C 180,E1 -3474.531,E2 -3474.531} C_VEL
LIN {X 0,Y 545.063,Z 44.595,A -85,B 0,C 180,E1 -3477.212,E2 -3477.212} C_VEL
LIN {X 0,Y 545.091,Z 44.697,A -85,B 0,C 180,E1 -3477.979,E2 -3477.979} C_VEL
LIN {X 0,Y 545.433,Z 49.599,A -85,B 0,C 180,E1 -3478.976,E2 -3478.976} C_VEL
LIN {X 0,Y 545.267,Z 62.352,A -85,B 0,C 180,E1 -3481.511,E2 -3481.511} C_VEL
LIN {X 0,Y 546.586,Z 69.729,A -85,B 0,C 180,E1 -3481.646,E2 -3481.646} C_VEL
LIN {X 0,Y 546.272,Z 168.418,A -85,B 0,C 180,E1 -3482.968,E2 -3482.968} C_VEL
LIN {X 0,Y 546.117,Z 181.152,A -85,B 0,C 180,E1 -3483.282,E2 -3483.282} C_VEL
LIN {X 0,Y 545.985,Z 193.621,A -85,B 0,C 180,E1 -3483.738,E2 -3483.738} C_VEL
LIN {X 0,Y 545.758,Z 205.858,A -85,B 0,C 180,E1 -3484.347,E2 -3484.347} C_VEL
LIN {X 0,Y 545.511,Z 216.671,A -85,B 0,C 180,E1 -3485.044,E2 -3485.044} C_VEL
LIN {X 0,Y 545.359,Z 226.322,A -85,B 0,C 180,E1 -3485.815,E2 -3485.815} C_VEL
LIN {X 0,Y 545.187,Z 234.929,A -85,B 0,C 180,E1 -3486.647,E2 -3486.647} C_VEL
LIN {X 0,Y 545.03,Z 243.41,A -85,B 0,C 180,E1 -3487.642,E2 -3487.642} C_VEL
LIN {X 0,Y 544.915,Z 249.613,A -85,B 0,C 180,E1 -3488.523,E2 -3488.523} C_VEL
LIN {X 0,Y 544.802,Z 255.989,A -85,B 0,C 180,E1 -3489.617,E2 -3489.617} C_VEL
LIN {X 0,Y 544.731,Z 261.436,A -85,B 0,C 180,E1 -3490.793,E2 -3490.793} C_VEL
LIN {X 0,Y 544.662,Z 265.578,A -85,B 0,C 180,E1 -3491.96,E2 -3491.96} C_VEL
LIN {X 0,Y 544.617,Z 267.675,A -85,B 0,C 180,E1 -3492.735,E2 -3492.735} C_VEL
LIN {X 0,Y 544.59,Z 269.325,A -85,B 0,C 180,E1 -3493.506,E2 -3493.506} C_VEL
LIN {X 0,Y 544.557,Z 270.538,A -85,B 0,C 180,E1 -3494.275,E2 -3494.275} C_VEL
LIN {X 0,Y 544.581,Z 271.528,A -85,B 0,C 180,E1 -3495.446,E2 -3495.446} C_VEL
LIN {X 0,Y 544.585,Z 271.549,A -85,B 0,C 180,E1 -3496.568,E2 -3496.568} C_VEL
LIN {X 0,Y 544.586,Z 271.055,A -85,B 0,C 180,E1 -3497.327,E2 -3497.327} C_VEL
LIN {X 0,Y 544.64,Z 269.033,A -85,B 0,C 180,E1 -3498.727,E2 -3498.727} C_VEL
LIN {X 0,Y 544.687,Z 266.022,A -85,B 0,C 180,E1 -3499.969,E2 -3499.969} C_VEL
LIN {X 0,Y 544.707,Z 262.211,A -85,B 0,C 180,E1 -3501.093,E2 -3501.093} C_VEL
LIN {X 0,Y 544.77,Z 257.278,A -85,B 0,C 180,E1 -3502.215,E2 -3502.215} C_VEL
LIN {X 0,Y 544.884,Z 251.084,A -85,B 0,C 180,E1 -3503.334,E2 -3503.334} C_VEL
LIN {X 0,Y 544.982,Z 243.373,A -85,B 0,C 180,E1 -3504.45,E2 -3504.45} C_VEL
LIN {X 0,Y 545.19,Z 233.75,A -85,B 0,C 180,E1 -3505.564,E2 -3505.564} C_VEL
LIN {X 0,Y 545.444,Z 223.795,A -85,B 0,C 180,E1 -3506.491,E2 -3506.491} C_VEL
LIN {X 0,Y 545.607,Z 213.981,A -85,B 0,C 180,E1 -3507.232,E2 -3507.232} C_VEL
LIN {X 0,Y 545.835,Z 203.319,A -85,B 0,C 180,E1 -3507.879,E2 -3507.879} C_VEL
LIN {X 0,Y 545.948,Z 191.674,A -85,B 0,C 180,E1 -3508.433,E2 -3508.433} C_VEL
LIN {X 0,Y 546.106,Z 179.097,A -85,B 0,C 180,E1 -3508.871,E2 -3508.871} C_VEL
LIN {X 0,Y 546.234,Z 166.968,A -85,B 0,C 180,E1 -3509.148,E2 -3509.148} C_VEL
LIN {X 0,Y 546.47,Z 68.617,A -85,B 0,C 180,E1 -3510.461,E2 -3510.461} C_VEL
LIN {X 0,Y 545.198,Z 62.117,A -85,B 0,C 180,E1 -3510.6,E2 -3510.6} C_VEL
LIN {X 0,Y 545.451,Z 48.462,A -85,B 0,C 180,E1 -3513.324,E2 -3513.324} C_VEL
LIN {X 0,Y 545.096,Z 44.588,A -85,B 0,C 180,E1 -3514.159,E2 -3514.159} C_VEL
LIN {X 0,Y 545.173,Z 44.573,A -85,B 0,C 180,E1 -3515.92,E2 -3515.92} C_VEL
LIN {X 0,Y 545.116,Z 44.583,A -85,B 0,C 180,E1 -3518.9,E2 -3518.9} C_VEL
LIN {X 0,Y 545.113,Z 44.58,A -85,B 0,C 180,E1 -3521.905,E2 -3521.905} C_VEL
LIN {X 0,Y 545.092,Z 44.583,A -85,B 0,C 180,E1 -3524.944,E2 -3524.944} C_VEL
LIN {X 0,Y 545.077,Z 44.588,A -85,B 0,C 180,E1 -3528.026,E2 -3528.026} C_VEL
LIN {X 0,Y 545.098,Z 44.587,A -85,B 0,C 180,E1 -3530.372,E2 -3530.372} C_VEL
LIN {X 0,Y 545.085,Z 44.584,A -85,B 0,C 180,E1 -3533.559,E2 -3533.559} C_VEL
LIN {X 0,Y 545.084,Z 44.591,A -85,B 0,C 180,E1 -3536.001,E2 -3536.001} C_VEL
LIN {X 0,Y 545.08,Z 44.583,A -85,B 0,C 180,E1 -3538.745,E2 -3538.745} C_VEL
LIN {X 0,Y 545.063,Z 44.591,A -85,B 0,C 180,E1 -3541.679,E2 -3541.679} C_VEL
LIN {X 0,Y 545.083,Z 44.582,A -85,B 0,C 180,E1 -3544.563,E2 -3544.563} C_VEL
LIN {X 0,Y 545.042,Z 44.591,A -85,B 0,C 180,E1 -3547.304,E2 -3547.304} C_VEL
LIN {X 0,Y 545.07,Z 44.585,A -85,B 0,C 180,E1 -3550.143,E2 -3550.143} C_VEL
LIN {X 0,Y 545.083,Z 44.586,A -85,B 0,C 180,E1 -3553.106,E2 -3553.106} C_VEL
LIN {X 0,Y 545.053,Z 44.586,A -85,B 0,C 180,E1 -3556.226,E2 -3556.226} C_VEL
LIN {X 0,Y 545.085,Z 44.586,A -85,B 0,C 180,E1 -3558.885,E2 -3558.885} C_VEL
LIN {X 0,Y 545.087,Z 44.586,A -85,B 0,C 180,E1 -3560.818,E2 -3560.818} C_VEL
LIN {X 0,Y 545.046,Z 44.588,A -85,B 0,C 180,E1 -3563.619,E2 -3563.619} C_VEL
LIN {X 0,Y 545.069,Z 44.585,A -85,B 0,C 180,E1 -3566.328,E2 -3566.328} C_VEL
LIN {X 0,Y 545.07,Z 44.592,A -85,B 0,C 180,E1 -3568.952,E2 -3568.952} C_VEL
LIN {X 0,Y 545.105,Z 44.58,A -85,B 0,C 180,E1 -3571.507,E2 -3571.507} C_VEL
LIN {X 0,Y 545.098,Z 44.586,A -85,B 0,C 180,E1 -3574.491,E2 -3574.491} C_VEL
LIN {X 0,Y 545.044,Z 44.588,A -85,B 0,C 180,E1 -3577.242,E2 -3577.242} C_VEL
LIN {X 0,Y 545.121,Z 44.586,A -85,B 0,C 180,E1 -3580.415,E2 -3580.415} C_VEL
LIN {X 0,Y 545.075,Z 44.583,A -85,B 0,C 180,E1 -3583.521,E2 -3583.521} C_VEL
LIN {X 0,Y 545.097,Z 44.583,A -85,B 0,C 180,E1 -3585.82,E2 -3585.82} C_VEL
LIN {X 0,Y 545.121,Z 44.578,A -85,B 0,C 180,E1 -3588.849,E2 -3588.849} C_VEL
LIN {X 0,Y 545.128,Z 44.582,A -85,B 0,C 180,E1 -3591.847,E2 -3591.847} C_VEL
LIN {X 0,Y 545.204,Z 44.567,A -85,B 0,C 180,E1 -3594.823,E2 -3594.823} C_VEL
LIN {X 0,Y 545.195,Z 44.576,A -85,B 0,C 180,E1 -3597.783,E2 -3597.783} C_VEL
LIN {X 0,Y 545.213,Z 44.566,A -85,B 0,C 180,E1 -3600.738,E2 -3600.738} C_VEL
LIN {X 0,Y 545.171,Z 44.572,A -85,B 0,C 180,E1 -3602.956,E2 -3602.956} C_VEL
LIN {X 0,Y 545.167,Z 44.576,A -85,B 0,C 180,E1 -3605.919,E2 -3605.919} C_VEL
LIN {X 0,Y 545.109,Z 44.58,A -85,B 0,C 180,E1 -3608.9,E2 -3608.9} C_VEL
LIN {X 0,Y 545.137,Z 44.577,A -85,B 0,C 180,E1 -3611.904,E2 -3611.904} C_VEL
LIN {X 0,Y 545.088,Z 44.586,A -85,B 0,C 180,E1 -3614.943,E2 -3614.943} C_VEL
LIN {X 0,Y 545.072,Z 44.583,A -85,B 0,C 180,E1 -3618.026,E2 -3618.026} C_VEL
LIN {X 0,Y 545.094,Z 44.581,A -85,B 0,C 180,E1 -3620.372,E2 -3620.372} C_VEL
LIN {X 0,Y 545.08,Z 44.584,A -85,B 0,C 180,E1 -3623.559,E2 -3623.559} C_VEL
LIN {X 0,Y 545.077,Z 44.583,A -85,B 0,C 180,E1 -3626.001,E2 -3626.001} C_VEL
LIN {X 0,Y 545.09,Z 44.59,A -85,B 0,C 180,E1 -3628.748,E2 -3628.748} C_VEL
LIN {X 0,Y 545.059,Z 44.585,A -85,B 0,C 180,E1 -3631.679,E2 -3631.679} C_VEL
LIN {X 0,Y 545.064,Z 44.594,A -85,B 0,C 180,E1 -3634.564,E2 -3634.564} C_VEL
LIN {X 0,Y 545.038,Z 44.588,A -85,B 0,C 180,E1 -3637.304,E2 -3637.304} C_VEL
LIN {X 0,Y 545.067,Z 44.59,A -85,B 0,C 180,E1 -3640.143,E2 -3640.143} C_VEL
LIN {X 0,Y 545.08,Z 44.583,A -85,B 0,C 180,E1 -3643.107,E2 -3643.107} C_VEL
LIN {X 0,Y 545.051,Z 44.594,A -85,B 0,C 180,E1 -3646.226,E2 -3646.226} C_VEL
LIN {X 0,Y 545.083,Z 44.582,A -85,B 0,C 180,E1 -3648.885,E2 -3648.885} C_VEL
LIN {X 0,Y 545.053,Z 44.592,A -85,B 0,C 180,E1 -3651.762,E2 -3651.762} C_VEL
LIN {X 0,Y 545.039,Z 44.589,A -85,B 0,C 180,E1 -3654.532,E2 -3654.532} C_VEL
LIN {X 0,Y 545.069,Z 44.585,A -85,B 0,C 180,E1 -3657.211,E2 -3657.211} C_VEL
LIN {X 0,Y 545.064,Z 44.593,A -85,B 0,C 180,E1 -3659.81,E2 -3659.81} C_VEL
LIN {X 0,Y 545.083,Z 44.585,A -85,B 0,C 180,E1 -3662.344,E2 -3662.344} C_VEL
LIN {X 0,Y 545.189,Z 44.757,A -85,B 0,C 180,E1 -3665.206,E2 -3665.206} C_VEL
LIN {X 0,Y 546.267,Z 51.721,A -85,B 0,C 180,E1 -3666.259,E2 -3666.259} C_VEL
LIN {X 0,Y 545.954,Z 70.05,A -85,B 0,C 180,E1 -3668.873,E2 -3668.873} C_VEL
LIN {X 0,Y 545.672,Z 90.886,A -85,B 0,C 180,E1 -3671.8,E2 -3671.8} C_VEL
LIN {X 0,Y 545.334,Z 113.071,A -85,B 0,C 180,E1 -3674.872,E2 -3674.872} C_VEL
LIN {X 0,Y 545.324,Z 117.31,A -85,B 0,C 180,E1 -3675.438,E2 -3675.438} C_VEL
LIN {X 0,Y 546.482,Z 126.701,A -85,B 0,C 180,E1 -3675.593,E2 -3675.593} C_VEL
LIN {X 0,Y 546.197,Z 225.791,A -85,B 0,C 180,E1 -3676.916,E2 -3676.916} C_VEL
LIN {X 0,Y 546.015,Z 238.367,A -85,B 0,C 180,E1 -3677.219,E2 -3677.219} C_VEL
LIN {X 0,Y 545.889,Z 251.349,A -85,B 0,C 180,E1 -3677.688,E2 -3677.688} C_VEL
LIN {X 0,Y 545.652,Z 262.772,A -85,B 0,C 180,E1 -3678.244,E2 -3678.244} C_VEL
LIN {X 0,Y 545.47,Z 274.021,A -85,B 0,C 180,E1 -3678.95,E2 -3678.95} C_VEL
LIN {X 0,Y 545.244,Z 284.731,A -85,B 0,C 180,E1 -3679.791,E2 -3679.791} C_VEL
LIN {X 0,Y 545.065,Z 294.387,A -85,B 0,C 180,E1 -3680.725,E2 -3680.725} C_VEL
LIN {X 0,Y 544.934,Z 302.306,A -85,B 0,C 180,E1 -3681.657,E2 -3681.657} C_VEL
LIN {X 0,Y 544.798,Z 310.041,A -85,B 0,C 180,E1 -3682.774,E2 -3682.774} C_VEL
LIN {X 0,Y 544.756,Z 317.176,A -85,B 0,C 180,E1 -3684.076,E2 -3684.076} C_VEL
LIN {X 0,Y 544.627,Z 321.918,A -85,B 0,C 180,E1 -3685.188,E2 -3685.188} C_VEL
LIN {X 0,Y 544.669,Z 325.549,A -85,B 0,C 180,E1 -3686.301,E2 -3686.301} C_VEL
LIN {X 0,Y 544.65,Z 327.419,A -85,B 0,C 180,E1 -3687.041,E2 -3687.041} C_VEL
LIN {X 0,Y 544.552,Z 329.819,A -85,B 0,C 180,E1 -3688.521,E2 -3688.521} C_VEL
LIN {X 0,Y 544.55,Z 330.43,A -85,B 0,C 180,E1 -3689.26,E2 -3689.26} C_VEL
LIN {X 0,Y 544.55,Z 330.647,A -85,B 0,C 180,E1 -3690,E2 -3690} C_VEL
LIN {X 0,Y 544.55,Z 330.43,A -85,B 0,C 180,E1 -3690.739,E2 -3690.739} C_VEL
LIN {X 0,Y 544.571,Z 328.82,A -85,B 0,C 180,E1 -3692.219,E2 -3692.219} C_VEL
LIN {X 0,Y 544.65,Z 327.42,A -85,B 0,C 180,E1 -3692.958,E2 -3692.958} C_VEL
LIN {X 0,Y 544.683,Z 324.47,A -85,B 0,C 180,E1 -3694.069,E2 -3694.069} C_VEL
LIN {X 0,Y 544.653,Z 320.472,A -85,B 0,C 180,E1 -3695.182,E2 -3695.182} C_VEL
LIN {X 0,Y 544.7,Z 315.189,A -85,B 0,C 180,E1 -3696.324,E2 -3696.324} C_VEL
LIN {X 0,Y 544.822,Z 308.863,A -85,B 0,C 180,E1 -3697.411,E2 -3697.411} C_VEL
LIN {X 0,Y 544.95,Z 300.794,A -85,B 0,C 180,E1 -3698.529,E2 -3698.529} C_VEL
LIN {X 0,Y 545.082,Z 292.574,A -85,B 0,C 180,E1 -3699.462,E2 -3699.462} C_VEL
LIN {X 0,Y 545.319,Z 282.557,A -85,B 0,C 180,E1 -3700.395,E2 -3700.395} C_VEL
LIN {X 0,Y 545.482,Z 271.677,A -85,B 0,C 180,E1 -3701.209,E2 -3701.209} C_VEL
LIN {X 0,Y 545.702,Z 260.173,A -85,B 0,C 180,E1 -3701.891,E2 -3701.891} C_VEL
LIN {X 0,Y 545.877,Z 247.905,A -85,B 0,C 180,E1 -3702.453,E2 -3702.453} C_VEL
LIN {X 0,Y 546.084,Z 235.034,A -85,B 0,C 180,E1 -3702.874,E2 -3702.874} C_VEL
LIN {X 0,Y 546.225,Z 222.89,A -85,B 0,C 180,E1 -3703.13,E2 -3703.13} C_VEL
LIN {X 0,Y 546.424,Z 125.198,A -85,B 0,C 180,E1 -3704.427,E2 -3704.427} C_VEL
LIN {X 0,Y 545.254,Z 116.984,A -85,B 0,C 180,E1 -3704.581,E2 -3704.581} C_VEL
LIN {X 0,Y 545.572,Z 95.993,A -85,B 0,C 180,E1 -3707.476,E2 -3707.476} C_VEL
LIN {X 0,Y 545.915,Z 75.48,A -85,B 0,C 180,E1 -3710.34,E2 -3710.34} C_VEL
LIN {X 0,Y 546.295,Z 51.573,A -85,B 0,C 180,E1 -3713.734,E2 -3713.734} C_VEL
LIN {X 0,Y 545.099,Z 44.588,A -85,B 0,C 180,E1 -3714.824,E2 -3714.824} C_VEL
LIN {X 0,Y 545.09,Z 44.585,A -85,B 0,C 180,E1 -3717.655,E2 -3717.655} C_VEL
LIN {X 0,Y 545.078,Z 44.592,A -85,B 0,C 180,E1 -3720.246,E2 -3720.246} C_VEL
LIN {X 0,Y 545.074,Z 44.585,A -85,B 0,C 180,E1 -3723.061,E2 -3723.061} C_VEL
LIN {X 0,Y 545.063,Z 44.589,A -85,B 0,C 180,E1 -3725.677,E2 -3725.677} C_VEL
LIN {X 0,Y 545.052,Z 44.591,A -85,B 0,C 180,E1 -3728.237,E2 -3728.237} C_VEL
LIN {X 0,Y 545.08,Z 44.584,A -85,B 0,C 180,E1 -3730.472,E2 -3730.472} C_VEL
LIN {X 0,Y 545.077,Z 44.585,A -85,B 0,C 180,E1 -3733.106,E2 -3733.106} C_VEL
LIN {X 0,Y 545.048,Z 44.587,A -85,B 0,C 180,E1 -3736.226,E2 -3736.226} C_VEL
LIN {X 0,Y 545.099,Z 44.582,A -85,B 0,C 180,E1 -3738.887,E2 -3738.887} C_VEL
LIN {X 0,Y 545.052,Z 44.588,A -85,B 0,C 180,E1 -3741.763,E2 -3741.763} C_VEL
LIN {X 0,Y 545.064,Z 44.586,A -85,B 0,C 180,E1 -3744.534,E2 -3744.534} C_VEL
LIN {X 0,Y 545.08,Z 44.591,A -85,B 0,C 180,E1 -3747.212,E2 -3747.212} C_VEL
LIN {X 0,Y 545.063,Z 44.585,A -85,B 0,C 180,E1 -3749.81,E2 -3749.81} C_VEL
LIN {X 0,Y 545.09,Z 44.583,A -85,B 0,C 180,E1 -3752.344,E2 -3752.344} C_VEL
LIN {X 0,Y 545.115,Z 44.587,A -85,B 0,C 180,E1 -3754.82,E2 -3754.82} C_VEL
LIN {X 0,Y 545.042,Z 44.587,A -85,B 0,C 180,E1 -3757.243,E2 -3757.243} C_VEL
LIN {X 0,Y 545.118,Z 44.585,A -85,B 0,C 180,E1 -3760.415,E2 -3760.415} C_VEL
LIN {X 0,Y 545.071,Z 44.583,A -85,B 0,C 180,E1 -3763.521,E2 -3763.521} C_VEL
LIN {X 0,Y 545.093,Z 44.583,A -85,B 0,C 180,E1 -3765.82,E2 -3765.82} C_VEL
LIN {X 0,Y 545.117,Z 44.579,A -85,B 0,C 180,E1 -3768.849,E2 -3768.849} C_VEL
LIN {X 0,Y 545.126,Z 44.582,A -85,B 0,C 180,E1 -3771.847,E2 -3771.847} C_VEL
LIN {X 0,Y 545.201,Z 44.568,A -85,B 0,C 180,E1 -3774.823,E2 -3774.823} C_VEL
LIN {X 0,Y 545.192,Z 44.575,A -85,B 0,C 180,E1 -3777.784,E2 -3777.784} C_VEL
LIN {X 0,Y 545.209,Z 44.567,A -85,B 0,C 180,E1 -3780.739,E2 -3780.739} C_VEL
LIN {X 0,Y 545.168,Z 44.57,A -85,B 0,C 180,E1 -3782.956,E2 -3782.956} C_VEL
LIN {X 0,Y 545.163,Z 44.575,A -85,B 0,C 180,E1 -3785.92,E2 -3785.92} C_VEL
LIN {X 0,Y 545.104,Z 44.58,A -85,B 0,C 180,E1 -3788.901,E2 -3788.901} C_VEL
LIN {X 0,Y 545.133,Z 44.576,A -85,B 0,C 180,E1 -3791.904,E2 -3791.904} C_VEL
LIN {X 0,Y 545.084,Z 44.588,A -85,B 0,C 180,E1 -3794.944,E2 -3794.944} C_VEL
LIN {X 0,Y 545.068,Z 44.583,A -85,B 0,C 180,E1 -3798.026,E2 -3798.026} C_VEL
LIN {X 0,Y 545.091,Z 44.584,A -85,B 0,C 180,E1 -3800.373,E2 -3800.373} C_VEL
LIN {X 0,Y 545.076,Z 44.584,A -85,B 0,C 180,E1 -3803.56,E2 -3803.56} C_VEL
LIN {X 0,Y 545.072,Z 44.583,A -85,B 0,C 180,E1 -3806.001,E2 -3806.001} C_VEL
LIN {X 0,Y 545.068,Z 44.589,A -85,B 0,C 180,E1 -3808.745,E2 -3808.745} C_VEL
LIN {X 0,Y 545.057,Z 44.587,A -85,B 0,C 180,E1 -3811.679,E2 -3811.679} C_VEL
LIN {X 0,Y 545.055,Z 44.59,A -85,B 0,C 180,E1 -3814.565,E2 -3814.565} C_VEL
LIN {X 0,Y 545.055,Z 44.587,A -85,B 0,C 180,E1 -3817,E2 -3817} C_VEL
LIN {X 0,Y 544.349,Z 44.678,A -85,B 0,C 180,E1 -3817.617,E2 -3817.617} C_VEL
LIN {X 0,Y 541.486,Z 45.034,A -85,B 0,C 180,E1 -3818.618,E2 -3818.618} C_VEL
LIN {X 0,Y 539.093,Z 45.333,A -85,B 0,C 180,E1 -3819.424,E2 -3819.424} C_VEL
LIN {X 0,Y 538.071,Z 45.463,A -85,B 0,C 180,E1 -3820.046,E2 -3820.046} C_VEL
LIN {X 0,Y 537.989,Z 45.467,A -85,B 0,C 180,E1 -3820.256,E2 -3820.256} C_VEL
LIN {X 0,Y 537.979,Z 45.47,A -85,B 0,C 180,E1 -3822.983,E2 -3822.983} C_VEL
LIN {X 0,Y 538.011,Z 45.473,A -85,B 0,C 180,E1 -3825.928,E2 -3825.928} C_VEL
LIN {X 0,Y 538.003,Z 45.468,A -85,B 0,C 180,E1 -3829.259,E2 -3829.259} C_VEL
LIN {X 0,Y 537.985,Z 45.47,A -85,B 0,C 180,E1 -3832.122,E2 -3832.122} C_VEL
LIN {X 0,Y 537.992,Z 45.471,A -85,B 0,C 180,E1 -3834.916,E2 -3834.916} C_VEL
LIN {X 0,Y 538.054,Z 45.516,A -85,B 0,C 180,E1 -3837.853,E2 -3837.853} C_VEL
LIN {X 0,Y 538.451,Z 50.922,A -85,B 0,C 180,E1 -3838.965,E2 -3838.965} C_VEL
LIN {X 0,Y 538.263,Z 62.607,A -85,B 0,C 180,E1 -3841.305,E2 -3841.305} C_VEL
LIN {X 0,Y 539.733,Z 70.446,A -85,B 0,C 180,E1 -3841.464,E2 -3841.464} C_VEL
LIN {X 0,Y 539.364,Z 168.693,A -85,B 0,C 180,E1 -3842.796,E2 -3842.796} C_VEL
LIN {X 0,Y 539.205,Z 181.695,A -85,B 0,C 180,E1 -3843.121,E2 -3843.121} C_VEL
LIN {X 0,Y 539.057,Z 194.121,A -85,B 0,C 180,E1 -3843.583,E2 -3843.583} C_VEL
LIN {X 0,Y 538.846,Z 205.508,A -85,B 0,C 180,E1 -3844.152,E2 -3844.152} C_VEL
LIN {X 0,Y 538.567,Z 217.13,A -85,B 0,C 180,E1 -3844.906,E2 -3844.906} C_VEL
LIN {X 0,Y 538.367,Z 227.147,A -85,B 0,C 180,E1 -3845.72,E2 -3845.72} C_VEL
LIN {X 0,Y 538.166,Z 237.234,A -85,B 0,C 180,E1 -3846.732,E2 -3846.732} C_VEL
LIN {X 0,Y 537.985,Z 245.325,A -85,B 0,C 180,E1 -3847.738,E2 -3847.738} C_VEL
LIN {X 0,Y 537.807,Z 253.131,A -85,B 0,C 180,E1 -3848.939,E2 -3848.939} C_VEL
LIN {X 0,Y 537.732,Z 259.708,A -85,B 0,C 180,E1 -3850.225,E2 -3850.225} C_VEL
LIN {X 0,Y 537.61,Z 264.062,A -85,B 0,C 180,E1 -3851.32,E2 -3851.32} C_VEL
LIN {X 0,Y 537.538,Z 267.938,A -85,B 0,C 180,E1 -3852.639,E2 -3852.639} C_VEL
LIN {X 0,Y 537.484,Z 270.654,A -85,B 0,C 180,E1 -3854.063,E2 -3854.063} C_VEL
LIN {X 0,Y 537.493,Z 271.879,A -85,B 0,C 180,E1 -3855.374,E2 -3855.374} C_VEL
LIN {X 0,Y 537.494,Z 271.973,A -85,B 0,C 180,E1 -3856.388,E2 -3856.388} C_VEL
LIN {X 0,Y 537.513,Z 271.593,A -85,B 0,C 180,E1 -3857.158,E2 -3857.158} C_VEL
LIN {X 0,Y 537.519,Z 270.793,A -85,B 0,C 180,E1 -3857.925,E2 -3857.925} C_VEL
LIN {X 0,Y 537.562,Z 269.552,A -85,B 0,C 180,E1 -3858.691,E2 -3858.691} C_VEL
LIN {X 0,Y 537.599,Z 266.923,A -85,B 0,C 180,E1 -3859.835,E2 -3859.835} C_VEL
LIN {X 0,Y 537.645,Z 263.28,A -85,B 0,C 180,E1 -3860.976,E2 -3860.976} C_VEL
LIN {X 0,Y 537.709,Z 258.531,A -85,B 0,C 180,E1 -3862.112,E2 -3862.112} C_VEL
LIN {X 0,Y 537.831,Z 252.359,A -85,B 0,C 180,E1 -3863.277,E2 -3863.277} C_VEL
LIN {X 0,Y 537.95,Z 245.112,A -85,B 0,C 180,E1 -3864.377,E2 -3864.377} C_VEL
LIN {X 0,Y 538.123,Z 237.54,A -85,B 0,C 180,E1 -3865.318,E2 -3865.318} C_VEL
LIN {X 0,Y 538.316,Z 228.369,A -85,B 0,C 180,E1 -3866.257,E2 -3866.257} C_VEL
LIN {X 0,Y 538.546,Z 218.186,A -85,B 0,C 180,E1 -3867.102,E2 -3867.102} C_VEL
LIN {X 0,Y 538.827,Z 206.899,A -85,B 0,C 180,E1 -3867.851,E2 -3867.851} C_VEL
LIN {X 0,Y 539.005,Z 195.204,A -85,B 0,C 180,E1 -3868.459,E2 -3868.459} C_VEL
LIN {X 0,Y 539.125,Z 182.315,A -85,B 0,C 180,E1 -3868.95,E2 -3868.95} C_VEL
LIN {X 0,Y 539.344,Z 169.443,A -85,B 0,C 180,E1 -3869.277,E2 -3869.277} C_VEL
LIN {X 0,Y 539.646,Z 82.32,A -85,B 0,C 180,E1 -3870.467,E2 -3870.467} C_VEL
LIN {X 0,Y 539.509,Z 68.816,A -85,B 0,C 180,E1 -3870.653,E2 -3870.653} C_VEL
LIN {X 0,Y 538.207,Z 62.435,A -85,B 0,C 180,E1 -3870.795,E2 -3870.795} C_VEL
LIN {X 0,Y 538.475,Z 49.633,A -85,B 0,C 180,E1 -3873.367,E2 -3873.367} C_VEL
LIN {X 0,Y 538.069,Z 45.464,A -85,B 0,C 180,E1 -3874.261,E2 -3874.261} C_VEL
LIN {X 0,Y 538.12,Z 45.458,A -85,B 0,C 180,E1 -3876.751,E2 -3876.751} C_VEL
LIN {X 0,Y 538.034,Z 45.46,A -85,B 0,C 180,E1 -3879.777,E2 -3879.777} C_VEL
LIN {X 0,Y 538.073,Z 45.458,A -85,B 0,C 180,E1 -3882.063,E2 -3882.063} C_VEL
LIN {X 0,Y 538.051,Z 45.459,A -85,B 0,C 180,E1 -3885.144,E2 -3885.144} C_VEL
LIN {X 0,Y 538.031,Z 45.469,A -85,B 0,C 180,E1 -3888.27,E2 -3888.27} C_VEL
LIN {X 0,Y 538.043,Z 45.462,A -85,B 0,C 180,E1 -3890.651,E2 -3890.651} C_VEL
LIN {X 0,Y 538.008,Z 45.469,A -85,B 0,C 180,E1 -3893.888,E2 -3893.888} C_VEL
LIN {X 0,Y 538.047,Z 45.463,A -85,B 0,C 180,E1 -3896.367,E2 -3896.367} C_VEL
LIN {X 0,Y 538.035,Z 45.46,A -85,B 0,C 180,E1 -3898.933,E2 -3898.933} C_VEL
LIN {X 0,Y 538.015,Z 45.471,A -85,B 0,C 180,E1 -3901.887,E2 -3901.887} C_VEL
LIN {X 0,Y 538.033,Z 45.46,A -85,B 0,C 180,E1 -3904.62,E2 -3904.62} C_VEL
LIN {X 0,Y 538.01,Z 45.466,A -85,B 0,C 180,E1 -3907.17,E2 -3907.17} C_VEL
LIN {X 0,Y 538.027,Z 45.466,A -85,B 0,C 180,E1 -3909.797,E2 -3909.797} C_VEL
LIN {X 0,Y 538.023,Z 45.463,A -85,B 0,C 180,E1 -3912.786,E2 -3912.786} C_VEL
LIN {X 0,Y 538.022,Z 45.463,A -85,B 0,C 180,E1 -3915.927,E2 -3915.927} C_VEL
LIN {X 0,Y 538.034,Z 45.46,A -85,B 0,C 180,E1 -3918.226,E2 -3918.226} C_VEL
LIN {X 0,Y 538.018,Z 45.471,A -85,B 0,C 180,E1 -3921.169,E2 -3921.169} C_VEL
LIN {X 0,Y 537.998,Z 45.465,A -85,B 0,C 180,E1 -3924.088,E2 -3924.088} C_VEL
LIN {X 0,Y 538.034,Z 45.466,A -85,B 0,C 180,E1 -3926.727,E2 -3926.727} C_VEL
LIN {X 0,Y 538.03,Z 45.461,A -85,B 0,C 180,E1 -3929.556,E2 -3929.556} C_VEL
LIN {X 0,Y 538.043,Z 45.459,A -85,B 0,C 180,E1 -3931.95,E2 -3931.95} C_VEL
LIN {X 0,Y 538.074,Z 45.461,A -85,B 0,C 180,E1 -3934.467,E2 -3934.467} C_VEL
LIN {X 0,Y 538.023,Z 45.466,A -85,B 0,C 180,E1 -3936.928,E2 -3936.928} C_VEL
LIN {X 0,Y 538.083,Z 45.458,A -85,B 0,C 180,E1 -3940.148,E2 -3940.148} C_VEL
LIN {X 0,Y 538.026,Z 45.461,A -85,B 0,C 180,E1 -3943.299,E2 -3943.299} C_VEL
LIN {X 0,Y 538.067,Z 45.457,A -85,B 0,C 180,E1 -3945.63,E2 -3945.63} C_VEL
LIN {X 0,Y 538.081,Z 45.456,A -85,B 0,C 180,E1 -3948.701,E2 -3948.701} C_VEL
LIN {X 0,Y 538.085,Z 45.458,A -85,B 0,C 180,E1 -3951.739,E2 -3951.739} C_VEL
LIN {X 0,Y 538.161,Z 45.445,A -85,B 0,C 180,E1 -3954.755,E2 -3954.755} C_VEL
LIN {X 0,Y 538.167,Z 45.451,A -85,B 0,C 180,E1 -3957.755,E2 -3957.755} C_VEL
LIN {X 0,Y 538.183,Z 45.441,A -85,B 0,C 180,E1 -3960.748,E2 -3960.748} C_VEL
LIN {X 0,Y 538.138,Z 45.448,A -85,B 0,C 180,E1 -3962.994,E2 -3962.994} C_VEL
LIN {X 0,Y 538.119,Z 45.453,A -85,B 0,C 180,E1 -3965.997,E2 -3965.997} C_VEL
LIN {X 0,Y 538.064,Z 45.457,A -85,B 0,C 180,E1 -3968.261,E2 -3968.261} C_VEL
LIN {X 0,Y 538.092,Z 45.459,A -85,B 0,C 180,E1 -3971.6,E2 -3971.6} C_VEL
LIN {X 0,Y 538.061,Z 45.46,A -85,B 0,C 180,E1 -3974.857,E2 -3974.857} C_VEL
LIN {X 0,Y 538.038,Z 45.463,A -85,B 0,C 180,E1 -3977.532,E2 -3977.532} C_VEL
LIN {X 0,Y 538.04,Z 45.463,A -85,B 0,C 180,E1 -3980.651,E2 -3980.651} C_VEL
LIN {X 0,Y 538.004,Z 45.464,A -85,B 0,C 180,E1 -3983.888,E2 -3983.888} C_VEL
LIN {X 0,Y 538.038,Z 45.462,A -85,B 0,C 180,E1 -3986.367,E2 -3986.367} C_VEL
LIN {X 0,Y 538.032,Z 45.467,A -85,B 0,C 180,E1 -3988.933,E2 -3988.933} C_VEL
LIN {X 0,Y 538.012,Z 45.463,A -85,B 0,C 180,E1 -3991.887,E2 -3991.887} C_VEL
LIN {X 0,Y 538.014,Z 45.471,A -85,B 0,C 180,E1 -3994.618,E2 -3994.618} C_VEL
LIN {X 0,Y 538.006,Z 45.464,A -85,B 0,C 180,E1 -3997.17,E2 -3997.17} C_VEL
LIN {X 0,Y 538.024,Z 45.463,A -85,B 0,C 180,E1 -3999.797,E2 -3999.797} C_VEL
LIN {X 0,Y 538.02,Z 45.464,A -85,B 0,C 180,E1 -4002.786,E2 -4002.786} C_VEL
LIN {X 0,Y 538.02,Z 45.467,A -85,B 0,C 180,E1 -4005.927,E2 -4005.927} C_VEL
LIN {X 0,Y 538.032,Z 45.467,A -85,B 0,C 180,E1 -4008.227,E2 -4008.227} C_VEL
LIN {X 0,Y 538.013,Z 45.463,A -85,B 0,C 180,E1 -4011.169,E2 -4011.169} C_VEL
LIN {X 0,Y 537.997,Z 45.471,A -85,B 0,C 180,E1 -4014.089,E2 -4014.089} C_VEL
LIN {X 0,Y 538.033,Z 45.46,A -85,B 0,C 180,E1 -4016.727,E2 -4016.727} C_VEL
LIN {X 0,Y 538.017,Z 45.469,A -85,B 0,C 180,E1 -4019.558,E2 -4019.558} C_VEL
LIN {X 0,Y 538.043,Z 45.466,A -85,B 0,C 180,E1 -4021.95,E2 -4021.95} C_VEL
LIN {X 0,Y 538.109,Z 45.598,A -85,B 0,C 180,E1 -4025.038,E2 -4025.038} C_VEL
LIN {X 0,Y 539.328,Z 52.995,A -85,B 0,C 180,E1 -4026.174,E2 -4026.174} C_VEL
LIN {X 0,Y 538.977,Z 71.082,A -85,B 0,C 180,E1 -4028.786,E2 -4028.786} C_VEL
LIN {X 0,Y 538.662,Z 91.91,A -85,B 0,C 180,E1 -4031.752,E2 -4031.752} C_VEL
LIN {X 0,Y 538.318,Z 112.687,A -85,B 0,C 180,E1 -4034.67,E2 -4034.67} C_VEL
LIN {X 0,Y 538.246,Z 116.751,A -85,B 0,C 180,E1 -4035.237,E2 -4035.237} C_VEL
LIN {X 0,Y 539.604,Z 126.885,A -85,B 0,C 180,E1 -4035.413,E2 -4035.413} C_VEL
LIN {X 0,Y 539.281,Z 225.376,A -85,B 0,C 180,E1 -4036.745,E2 -4036.745} C_VEL
LIN {X 0,Y 539.072,Z 238.728,A -85,B 0,C 180,E1 -4037.075,E2 -4037.075} C_VEL
LIN {X 0,Y 538.921,Z 250.95,A -85,B 0,C 180,E1 -4037.526,E2 -4037.526} C_VEL
LIN {X 0,Y 538.66,Z 262.736,A -85,B 0,C 180,E1 -4038.109,E2 -4038.109} C_VEL
LIN {X 0,Y 538.424,Z 274.929,A -85,B 0,C 180,E1 -4038.899,E2 -4038.899} C_VEL
LIN {X 0,Y 538.189,Z 285.418,A -85,B 0,C 180,E1 -4039.751,E2 -4039.751} C_VEL
LIN {X 0,Y 538.022,Z 293.999,A -85,B 0,C 180,E1 -4040.602,E2 -4040.602} C_VEL
LIN {X 0,Y 537.876,Z 301.919,A -85,B 0,C 180,E1 -4041.547,E2 -4041.547} C_VEL
LIN {X 0,Y 537.711,Z 309.655,A -85,B 0,C 180,E1 -4042.678,E2 -4042.678} C_VEL
LIN {X 0,Y 537.644,Z 316.79,A -85,B 0,C 180,E1 -4043.997,E2 -4043.997} C_VEL
LIN {X 0,Y 537.539,Z 321.535,A -85,B 0,C 180,E1 -4045.125,E2 -4045.125} C_VEL
LIN {X 0,Y 537.591,Z 325.166,A -85,B 0,C 180,E1 -4046.252,E2 -4046.252} C_VEL
LIN {X 0,Y 537.58,Z 327.037,A -85,B 0,C 180,E1 -4047.002,E2 -4047.002} C_VEL
LIN {X 0,Y 537.461,Z 329.436,A -85,B 0,C 180,E1 -4048.501,E2 -4048.501} C_VEL
LIN {X 0,Y 537.46,Z 330.046,A -85,B 0,C 180,E1 -4049.25,E2 -4049.25} C_VEL
LIN {X 0,Y 537.461,Z 330.263,A -85,B 0,C 180,E1 -4050,E2 -4050} C_VEL
LIN {X 0,Y 537.46,Z 330.045,A -85,B 0,C 180,E1 -4050.749,E2 -4050.749} C_VEL
LIN {X 0,Y 537.49,Z 328.434,A -85,B 0,C 180,E1 -4052.248,E2 -4052.248} C_VEL
LIN {X 0,Y 537.58,Z 327.034,A -85,B 0,C 180,E1 -4052.997,E2 -4052.997} C_VEL
LIN {X 0,Y 537.602,Z 324.081,A -85,B 0,C 180,E1 -4054.123,E2 -4054.123} C_VEL
LIN {X 0,Y 537.587,Z 320.082,A -85,B 0,C 180,E1 -4055.25,E2 -4055.25} C_VEL
LIN {X 0,Y 537.64,Z 314.026,A -85,B 0,C 180,E1 -4056.551,E2 -4056.551} C_VEL
LIN {X 0,Y 537.749,Z 307.223,A -85,B 0,C 180,E1 -4057.698,E2 -4057.698} C_VEL
LIN {X 0,Y 537.909,Z 298.896,A -85,B 0,C 180,E1 -4058.831,E2 -4058.831} C_VEL
LIN {X 0,Y 538.057,Z 290.362,A -85,B 0,C 180,E1 -4059.776,E2 -4059.776} C_VEL
LIN {X 0,Y 538.293,Z 279.825,A -85,B 0,C 180,E1 -4060.722,E2 -4060.722} C_VEL
LIN {X 0,Y 538.52,Z 268.724,A -85,B 0,C 180,E1 -4061.525,E2 -4061.525} C_VEL
LIN {X 0,Y 538.777,Z 257.988,A -85,B 0,C 180,E1 -4062.142,E2 -4062.142} C_VEL
LIN {X 0,Y 538.973,Z 246.269,A -85,B 0,C 180,E1 -4062.663,E2 -4062.663} C_VEL
LIN {X 0,Y 539.167,Z 232.774,A -85,B 0,C 180,E1 -4063.09,E2 -4063.09} C_VEL
LIN {X 0,Y 539.353,Z 219.406,A -85,B 0,C 180,E1 -4063.349,E2 -4063.349} C_VEL
LIN {X 0,Y 539.46,Z 125.393,A -85,B 0,C 180,E1 -4064.61,E2 -4064.61} C_VEL
LIN {X 0,Y 538.25,Z 116.521,A -85,B 0,C 180,E1 -4064.783,E2 -4064.783} C_VEL
LIN {X 0,Y 538.575,Z 95.576,A -85,B 0,C 180,E1 -4067.712,E2 -4067.712} C_VEL
LIN {X 0,Y 538.937,Z 76.192,A -85,B 0,C 180,E1 -4070.458,E2 -4070.458} C_VEL
LIN {X 0,Y 539.36,Z 52.822,A -85,B 0,C 180,E1 -4073.824,E2 -4073.824} C_VEL
LIN {X 0,Y 538.062,Z 45.464,A -85,B 0,C 180,E1 -4074.964,E2 -4074.964} C_VEL
LIN {X 0,Y 538.045,Z 45.466,A -85,B 0,C 180,E1 -4078.049,E2 -4078.049} C_VEL
LIN {X 0,Y 538.021,Z 45.468,A -85,B 0,C 180,E1 -4080.626,E2 -4080.626} C_VEL
LIN {X 0,Y 538.019,Z 45.464,A -85,B 0,C 180,E1 -4083.278,E2 -4083.278} C_VEL
LIN {X 0,Y 538.028,Z 45.469,A -85,B 0,C 180,E1 -4086.002,E2 -4086.002} C_VEL
LIN {X 0,Y 538.012,Z 45.464,A -85,B 0,C 180,E1 -4088.83,E2 -4088.83} C_VEL
LIN {X 0,Y 538.029,Z 45.469,A -85,B 0,C 180,E1 -4091.773,E2 -4091.773} C_VEL
LIN {X 0,Y 538.005,Z 45.463,A -85,B 0,C 180,E1 -4094.862,E2 -4094.862} C_VEL
LIN {X 0,Y 538.036,Z 45.462,A -85,B 0,C 180,E1 -4098.12,E2 -4098.12} C_VEL
LIN {X 0,Y 538.058,Z 45.458,A -85,B 0,C 180,E1 -4100.411,E2 -4100.411} C_VEL
LIN {X 0,Y 538.028,Z 45.466,A -85,B 0,C 180,E1 -4103.067,E2 -4103.067} C_VEL
LIN {X 0,Y 538.026,Z 45.462,A -85,B 0,C 180,E1 -4105.827,E2 -4105.827} C_VEL
LIN {X 0,Y 538.008,Z 45.466,A -85,B 0,C 180,E1 -4108.499,E2 -4108.499} C_VEL
LIN {X 0,Y 538.058,Z 45.464,A -85,B 0,C 180,E1 -4111.1,E2 -4111.1} C_VEL
LIN {X 0,Y 538.04,Z 45.459,A -85,B 0,C 180,E1 -4113.633,E2 -4113.633} C_VEL
LIN {X 0,Y 538.021,Z 45.463,A -85,B 0,C 180,E1 -4116.118,E2 -4116.118} C_VEL
LIN {X 0,Y 538.038,Z 45.461,A -85,B 0,C 180,E1 -4119.349,E2 -4119.349} C_VEL
LIN {X 0,Y 538.052,Z 45.464,A -85,B 0,C 180,E1 -4122.517,E2 -4122.517} C_VEL
LIN {X 0,Y 538.062,Z 45.458,A -85,B 0,C 180,E1 -4125.631,E2 -4125.631} C_VEL
LIN {X 0,Y 538.076,Z 45.458,A -85,B 0,C 180,E1 -4128.702,E2 -4128.702} C_VEL
LIN {X 0,Y 538.084,Z 45.458,A -85,B 0,C 180,E1 -4131.74,E2 -4131.74} C_VEL
LIN {X 0,Y 538.159,Z 45.445,A -85,B 0,C 180,E1 -4134.755,E2 -4134.755} C_VEL
LIN {X 0,Y 538.164,Z 45.45,A -85,B 0,C 180,E1 -4137.755,E2 -4137.755} C_VEL
LIN {X 0,Y 538.18,Z 45.442,A -85,B 0,C 180,E1 -4140.748,E2 -4140.748} C_VEL
LIN {X 0,Y 538.135,Z 45.447,A -85,B 0,C 180,E1 -4142.995,E2 -4142.995} C_VEL
LIN {X 0,Y 538.115,Z 45.452,A -85,B 0,C 180,E1 -4145.998,E2 -4145.998} C_VEL
LIN {X 0,Y 538.057,Z 45.459,A -85,B 0,C 180,E1 -4149.018,E2 -4149.018} C_VEL
LIN {X 0,Y 538.081,Z 45.454,A -85,B 0,C 180,E1 -4152.063,E2 -4152.063} C_VEL
LIN {X 0,Y 538.044,Z 45.468,A -85,B 0,C 180,E1 -4155.144,E2 -4155.144} C_VEL
LIN {X 0,Y 538.023,Z 45.461,A -85,B 0,C 180,E1 -4158.271,E2 -4158.271} C_VEL
LIN {X 0,Y 538.036,Z 45.466,A -85,B 0,C 180,E1 -4160.652,E2 -4160.652} C_VEL
LIN {X 0,Y 538,Z 45.465,A -85,B 0,C 180,E1 -4163.889,E2 -4163.889} C_VEL
LIN {X 0,Y 538.033,Z 45.464,A -85,B 0,C 180,E1 -4166.367,E2 -4166.367} C_VEL
LIN {X 0,Y 538.029,Z 45.463,A -85,B 0,C 180,E1 -4168.934,E2 -4168.934} C_VEL
LIN {X 0,Y 538.009,Z 45.466,A -85,B 0,C 180,E1 -4171.888,E2 -4171.888} C_VEL
LIN {X 0,Y 538.004,Z 45.467,A -85,B 0,C 180,E1 -4174.617,E2 -4174.617} C_VEL
LIN {X 0,Y 537.998,Z 45.465,A -85,B 0,C 180,E1 -4177.17,E2 -4177.17} C_VEL
LIN {X 0,Y 538.01,Z 45.47,A -85,B 0,C 180,E1 -4179.799,E2 -4179.799} C_VEL
LIN {X 0,Y 537.989,Z 45.467,A -85,B 0,C 180,E1 -4180.256,E2 -4180.256} C_VEL
LIN {X 0,Y 537.326,Z 45.548,A -85,B 0,C 180,E1 -4180.881,E2 -4180.881} C_VEL
LIN {X 0,Y 534.469,Z 45.91,A -85,B 0,C 180,E1 -4181.896,E2 -4181.896} C_VEL
LIN {X 0,Y 532.052,Z 46.215,A -85,B 0,C 180,E1 -4182.713,E2 -4182.713} C_VEL
LIN {X 0,Y 531.012,Z 46.342,A -85,B 0,C 180,E1 -4183.344,E2 -4183.344} C_VEL
LIN {X 0,Y 530.927,Z 46.351,A -85,B 0,C 180,E1 -4183.558,E2 -4183.558} C_VEL
LIN {X 0,Y 530.938,Z 46.348,A -85,B 0,C 180,E1 -4186.503,E2 -4186.503} C_VEL
LIN {X 0,Y 530.948,Z 46.352,A -85,B 0,C 180,E1 -4189.565,E2 -4189.565} C_VEL
LIN {X 0,Y 530.939,Z 46.346,A -85,B 0,C 180,E1 -4192.582,E2 -4192.582} C_VEL
LIN {X 0,Y 530.977,Z 46.349,A -85,B 0,C 180,E1 -4195.31,E2 -4195.31} C_VEL
LIN {X 0,Y 531.019,Z 46.473,A -85,B 0,C 180,E1 -4197.749,E2 -4197.749} C_VEL
LIN {X 0,Y 531.486,Z 51.208,A -85,B 0,C 180,E1 -4198.734,E2 -4198.734} C_VEL
LIN {X 0,Y 531.271,Z 63.042,A -85,B 0,C 180,E1 -4201.118,E2 -4201.118} C_VEL
LIN {X 0,Y 532.9,Z 71.315,A -85,B 0,C 180,E1 -4201.279,E2 -4201.279} C_VEL
LIN {X 0,Y 532.486,Z 168.984,A -85,B 0,C 180,E1 -4202.621,E2 -4202.621} C_VEL
LIN {X 0,Y 532.303,Z 182.243,A -85,B 0,C 180,E1 -4202.956,E2 -4202.956} C_VEL
LIN {X 0,Y 532.13,Z 195.416,A -85,B 0,C 180,E1 -4203.458,E2 -4203.458} C_VEL
LIN {X 0,Y 531.893,Z 206.825,A -85,B 0,C 180,E1 -4204.051,E2 -4204.051} C_VEL
LIN {X 0,Y 531.613,Z 217.584,A -85,B 0,C 180,E1 -4204.764,E2 -4204.764} C_VEL
LIN {X 0,Y 531.372,Z 228.724,A -85,B 0,C 180,E1 -4205.691,E2 -4205.691} C_VEL
LIN {X 0,Y 531.153,Z 237.661,A -85,B 0,C 180,E1 -4206.613,E2 -4206.613} C_VEL
LIN {X 0,Y 530.943,Z 246.351,A -85,B 0,C 180,E1 -4207.719,E2 -4207.719} C_VEL
LIN {X 0,Y 530.761,Z 253.546,A -85,B 0,C 180,E1 -4208.849,E2 -4208.849} C_VEL
LIN {X 0,Y 530.691,Z 259.871,A -85,B 0,C 180,E1 -4210.097,E2 -4210.097} C_VEL
LIN {X 0,Y 530.532,Z 265.113,A -85,B 0,C 180,E1 -4211.463,E2 -4211.463} C_VEL
LIN {X 0,Y 530.472,Z 268.191,A -85,B 0,C 180,E1 -4212.536,E2 -4212.536} C_VEL
LIN {X 0,Y 530.402,Z 270.759,A -85,B 0,C 180,E1 -4213.844,E2 -4213.844} C_VEL
LIN {X 0,Y 530.411,Z 272.222,A -85,B 0,C 180,E1 -4215.3,E2 -4215.3} C_VEL
LIN {X 0,Y 530.419,Z 272.396,A -85,B 0,C 180,E1 -4216.202,E2 -4216.202} C_VEL
LIN {X 0,Y 530.433,Z 272.095,A -85,B 0,C 180,E1 -4216.983,E2 -4216.983} C_VEL
LIN {X 0,Y 530.447,Z 271.401,A -85,B 0,C 180,E1 -4217.761,E2 -4217.761} C_VEL
LIN {X 0,Y 530.49,Z 270.117,A -85,B 0,C 180,E1 -4218.629,E2 -4218.629} C_VEL
LIN {X 0,Y 530.536,Z 266.754,A -85,B 0,C 180,E1 -4220.084,E2 -4220.084} C_VEL
LIN {X 0,Y 530.584,Z 262.929,A -85,B 0,C 180,E1 -4221.239,E2 -4221.239} C_VEL
LIN {X 0,Y 530.677,Z 257.982,A -85,B 0,C 180,E1 -4222.39,E2 -4222.39} C_VEL
LIN {X 0,Y 530.81,Z 252.044,A -85,B 0,C 180,E1 -4223.492,E2 -4223.492} C_VEL
LIN {X 0,Y 530.938,Z 244.045,A -85,B 0,C 180,E1 -4224.684,E2 -4224.684} C_VEL
LIN {X 0,Y 531.21,Z 234.396,A -85,B 0,C 180,E1 -4225.827,E2 -4225.827} C_VEL
LIN {X 0,Y 531.497,Z 224.411,A -85,B 0,C 180,E1 -4226.779,E2 -4226.779} C_VEL
LIN {X 0,Y 531.701,Z 214.561,A -85,B 0,C 180,E1 -4227.538,E2 -4227.538} C_VEL
LIN {X 0,Y 532.002,Z 202.119,A -85,B 0,C 180,E1 -4228.297,E2 -4228.297} C_VEL
LIN {X 0,Y 532.197,Z 189.829,A -85,B 0,C 180,E1 -4228.865,E2 -4228.865} C_VEL
LIN {X 0,Y 532.353,Z 177.627,A -85,B 0,C 180,E1 -4229.267,E2 -4229.267} C_VEL
LIN {X 0,Y 532.493,Z 163.973,A -85,B 0,C 180,E1 -4229.551,E2 -4229.551} C_VEL
LIN {X 0,Y 532.771,Z 70.3,A -85,B 0,C 180,E1 -4230.827,E2 -4230.827} C_VEL
LIN {X 0,Y 531.218,Z 62.761,A -85,B 0,C 180,E1 -4230.995,E2 -4230.995} C_VEL
LIN {X 0,Y 531.496,Z 50.804,A -85,B 0,C 180,E1 -4233.412,E2 -4233.412} C_VEL
LIN {X 0,Y 531.036,Z 46.34,A -85,B 0,C 180,E1 -4234.365,E2 -4234.365} C_VEL
LIN {X 0,Y 531.081,Z 46.334,A -85,B 0,C 180,E1 -4236.84,E2 -4236.84} C_VEL
LIN {X 0,Y 531.026,Z 46.335,A -85,B 0,C 180,E1 -4239.138,E2 -4239.138} C_VEL
LIN {X 0,Y 531.036,Z 46.336,A -85,B 0,C 180,E1 -4242.225,E2 -4242.225} C_VEL
LIN {X 0,Y 531.001,Z 46.336,A -85,B 0,C 180,E1 -4245.35,E2 -4245.35} C_VEL
LIN {X 0,Y 530.991,Z 46.343,A -85,B 0,C 180,E1 -4248.521,E2 -4248.521} C_VEL
LIN {X 0,Y 531.005,Z 46.336,A -85,B 0,C 180,E1 -4250.938,E2 -4250.938} C_VEL
LIN {X 0,Y 530.971,Z 46.347,A -85,B 0,C 180,E1 -4254.225,E2 -4254.225} C_VEL
LIN {X 0,Y 531.01,Z 46.336,A -85,B 0,C 180,E1 -4256.744,E2 -4256.744} C_VEL
LIN {X 0,Y 530.986,Z 46.34,A -85,B 0,C 180,E1 -4259.323,E2 -4259.323} C_VEL
LIN {X 0,Y 530.971,Z 46.345,A -85,B 0,C 180,E1 -4262.1,E2 -4262.1} C_VEL
LIN {X 0,Y 530.989,Z 46.338,A -85,B 0,C 180,E1 -4264.853,E2 -4264.853} C_VEL
LIN {X 0,Y 530.97,Z 46.347,A -85,B 0,C 180,E1 -4267.508,E2 -4267.508} C_VEL
LIN {X 0,Y 530.985,Z 46.338,A -85,B 0,C 180,E1 -4270.433,E2 -4270.433} C_VEL
LIN {X 0,Y 530.965,Z 46.347,A -85,B 0,C 180,E1 -4273.281,E2 -4273.281} C_VEL
LIN {X 0,Y 530.98,Z 46.344,A -85,B 0,C 180,E1 -4275.622,E2 -4275.622} C_VEL
LIN {X 0,Y 530.997,Z 46.338,A -85,B 0,C 180,E1 -4278.564,E2 -4278.564} C_VEL
LIN {X 0,Y 530.962,Z 46.345,A -85,B 0,C 180,E1 -4281.529,E2 -4281.529} C_VEL
LIN {X 0,Y 530.959,Z 46.342,A -85,B 0,C 180,E1 -4284.38,E2 -4284.38} C_VEL
LIN {X 0,Y 530.97,Z 46.346,A -85,B 0,C 180,E1 -4287.133,E2 -4287.133} C_VEL
LIN {X 0,Y 530.973,Z 46.34,A -85,B 0,C 180,E1 -4289.803,E2 -4289.803} C_VEL
LIN {X 0,Y 531.016,Z 46.339,A -85,B 0,C 180,E1 -4292.467,E2 -4292.467} C_VEL
LIN {X 0,Y 531.009,Z 46.34,A -85,B 0,C 180,E1 -4294.942,E2 -4294.942} C_VEL
LIN {X 0,Y 530.975,Z 46.344,A -85,B 0,C 180,E1 -4298.246,E2 -4298.246} C_VEL
LIN {X 0,Y 530.996,Z 46.343,A -85,B 0,C 180,E1 -4300.677,E2 -4300.677} C_VEL
LIN {X 0,Y 530.988,Z 46.339,A -85,B 0,C 180,E1 -4303.071,E2 -4303.071} C_VEL
LIN {X 0,Y 531.022,Z 46.334,A -85,B 0,C 180,E1 -4305.436,E2 -4305.436} C_VEL
LIN {X 0,Y 531.04,Z 46.335,A -85,B 0,C 180,E1 -4308.55,E2 -4308.55} C_VEL
LIN {X 0,Y 531.055,Z 46.332,A -85,B 0,C 180,E1 -4311.629,E2 -4311.629} C_VEL
LIN {X 0,Y 531.121,Z 46.322,A -85,B 0,C 180,E1 -4314.685,E2 -4314.685} C_VEL
LIN {X 0,Y 531.14,Z 46.326,A -85,B 0,C 180,E1 -4317.725,E2 -4317.725} C_VEL
LIN {X 0,Y 531.154,Z 46.317,A -85,B 0,C 180,E1 -4320.758,E2 -4320.758} C_VEL
LIN {X 0,Y 531.105,Z 46.324,A -85,B 0,C 180,E1 -4323.034,E2 -4323.034} C_VEL
LIN {X 0,Y 531.075,Z 46.329,A -85,B 0,C 180,E1 -4326.077,E2 -4326.077} C_VEL
LIN {X 0,Y 531.024,Z 46.338,A -85,B 0,C 180,E1 -4329.138,E2 -4329.138} C_VEL
LIN {X 0,Y 531.042,Z 46.331,A -85,B 0,C 180,E1 -4332.225,E2 -4332.225} C_VEL
LIN {X 0,Y 530.998,Z 46.344,A -85,B 0,C 180,E1 -4335.35,E2 -4335.35} C_VEL
LIN {X 0,Y 530.987,Z 46.339,A -85,B 0,C 180,E1 -4338.521,E2 -4338.521} C_VEL
LIN {X 0,Y 531.001,Z 46.344,A -85,B 0,C 180,E1 -4340.938,E2 -4340.938} C_VEL
LIN {X 0,Y 530.971,Z 46.341,A -85,B 0,C 180,E1 -4344.225,E2 -4344.225} C_VEL
LIN {X 0,Y 530.991,Z 46.345,A -85,B 0,C 180,E1 -4346.744,E2 -4346.744} C_VEL
LIN {X 0,Y 530.983,Z 46.34,A -85,B 0,C 180,E1 -4349.323,E2 -4349.323} C_VEL
LIN {X 0,Y 530.967,Z 46.342,A -85,B 0,C 180,E1 -4352.1,E2 -4352.1} C_VEL
LIN {X 0,Y 530.972,Z 46.345,A -85,B 0,C 180,E1 -4354.851,E2 -4354.851} C_VEL
LIN {X 0,Y 530.967,Z 46.34,A -85,B 0,C 180,E1 -4357.508,E2 -4357.508} C_VEL
LIN {X 0,Y 530.983,Z 46.347,A -85,B 0,C 180,E1 -4360.433,E2 -4360.433} C_VEL
LIN {X 0,Y 530.962,Z 46.341,A -85,B 0,C 180,E1 -4363.281,E2 -4363.281} C_VEL
LIN {X 0,Y 530.978,Z 46.341,A -85,B 0,C 180,E1 -4365.622,E2 -4365.622} C_VEL
LIN {X 0,Y 530.995,Z 46.339,A -85,B 0,C 180,E1 -4368.564,E2 -4368.564} C_VEL
LIN {X 0,Y 530.957,Z 46.344,A -85,B 0,C 180,E1 -4371.529,E2 -4371.529} C_VEL
LIN {X 0,Y 530.957,Z 46.344,A -85,B 0,C 180,E1 -4374.38,E2 -4374.38} C_VEL
LIN {X 0,Y 530.969,Z 46.341,A -85,B 0,C 180,E1 -4377.133,E2 -4377.133} C_VEL
LIN {X 0,Y 530.964,Z 46.35,A -85,B 0,C 180,E1 -4379.802,E2 -4379.802} C_VEL
LIN {X 0,Y 531.015,Z 46.338,A -85,B 0,C 180,E1 -4382.468,E2 -4382.468} C_VEL
LIN {X 0,Y 531.06,Z 46.417,A -85,B 0,C 180,E1 -4384.866,E2 -4384.866} C_VEL
LIN {X 0,Y 532.37,Z 54.008,A -85,B 0,C 180,E1 -4386.05,E2 -4386.05} C_VEL
LIN {X 0,Y 532.017,Z 72.11,A -85,B 0,C 180,E1 -4388.698,E2 -4388.698} C_VEL
LIN {X 0,Y 531.67,Z 92.895,A -85,B 0,C 180,E1 -4391.698,E2 -4391.698} C_VEL
LIN {X 0,Y 531.287,Z 113.687,A -85,B 0,C 180,E1 -4394.659,E2 -4394.659} C_VEL
LIN {X 0,Y 531.207,Z 116.347,A -85,B 0,C 180,E1 -4395.034,E2 -4395.034} C_VEL
LIN {X 0,Y 532.736,Z 128.157,A -85,B 0,C 180,E1 -4395.243,E2 -4395.243} C_VEL
LIN {X 0,Y 532.387,Z 224.962,A -85,B 0,C 180,E1 -4396.57,E2 -4396.57} C_VEL
LIN {X 0,Y 532.15,Z 238.325,A -85,B 0,C 180,E1 -4396.904,E2 -4396.904} C_VEL
LIN {X 0,Y 531.952,Z 250.551,A -85,B 0,C 180,E1 -4397.36,E2 -4397.36} C_VEL
LIN {X 0,Y 531.662,Z 262.615,A -85,B 0,C 180,E1 -4397.967,E2 -4397.967} C_VEL
LIN {X 0,Y 531.43,Z 274.538,A -85,B 0,C 180,E1 -4398.751,E2 -4398.751} C_VEL
LIN {X 0,Y 531.191,Z 285.03,A -85,B 0,C 180,E1 -4399.614,E2 -4399.614} C_VEL
LIN {X 0,Y 530.958,Z 293.61,A -85,B 0,C 180,E1 -4400.476,E2 -4400.476} C_VEL
LIN {X 0,Y 530.784,Z 301.53,A -85,B 0,C 180,E1 -4401.433,E2 -4401.433} C_VEL
LIN {X 0,Y 530.642,Z 309.27,A -85,B 0,C 180,E1 -4402.58,E2 -4402.58} C_VEL
LIN {X 0,Y 530.537,Z 316.405,A -85,B 0,C 180,E1 -4403.916,E2 -4403.916} C_VEL
LIN {X 0,Y 530.458,Z 321.151,A -85,B 0,C 180,E1 -4405.059,E2 -4405.059} C_VEL
LIN {X 0,Y 530.516,Z 324.784,A -85,B 0,C 180,E1 -4406.202,E2 -4406.202} C_VEL
LIN {X 0,Y 530.512,Z 326.656,A -85,B 0,C 180,E1 -4406.962,E2 -4406.962} C_VEL
LIN {X 0,Y 530.37,Z 329.053,A -85,B 0,C 180,E1 -4408.481,E2 -4408.481} C_VEL
LIN {X 0,Y 530.369,Z 329.663,A -85,B 0,C 180,E1 -4409.24,E2 -4409.24} C_VEL
LIN {X 0,Y 530.372,Z 329.879,A -85,B 0,C 180,E1 -4410,E2 -4410} C_VEL
LIN {X 0,Y 530.37,Z 329.661,A -85,B 0,C 180,E1 -4410.759,E2 -4410.759} C_VEL
LIN {X 0,Y 530.412,Z 328.048,A -85,B 0,C 180,E1 -4412.278,E2 -4412.278} C_VEL
LIN {X 0,Y 530.512,Z 326.648,A -85,B 0,C 180,E1 -4413.037,E2 -4413.037} C_VEL
LIN {X 0,Y 530.521,Z 323.693,A -85,B 0,C 180,E1 -4414.178,E2 -4414.178} C_VEL
LIN {X 0,Y 530.52,Z 319.692,A -85,B 0,C 180,E1 -4415.32,E2 -4415.32} C_VEL
LIN {X 0,Y 530.538,Z 314.24,A -85,B 0,C 180,E1 -4416.525,E2 -4416.525} C_VEL
LIN {X 0,Y 530.659,Z 308.07,A -85,B 0,C 180,E1 -4417.61,E2 -4417.61} C_VEL
LIN {X 0,Y 530.81,Z 299.996,A -85,B 0,C 180,E1 -4418.758,E2 -4418.758} C_VEL
LIN {X 0,Y 530.969,Z 291.77,A -85,B 0,C 180,E1 -4419.715,E2 -4419.715} C_VEL
LIN {X 0,Y 531.262,Z 281.749,A -85,B 0,C 180,E1 -4420.673,E2 -4420.673} C_VEL
LIN {X 0,Y 531.461,Z 270.354,A -85,B 0,C 180,E1 -4421.542,E2 -4421.542} C_VEL
LIN {X 0,Y 531.762,Z 259.353,A -85,B 0,C 180,E1 -4422.208,E2 -4422.208} C_VEL
LIN {X 0,Y 532.017,Z 247.078,A -85,B 0,C 180,E1 -4422.783,E2 -4422.783} C_VEL
LIN {X 0,Y 532.265,Z 234.184,A -85,B 0,C 180,E1 -4423.214,E2 -4423.214} C_VEL
LIN {X 0,Y 532.438,Z 222.005,A -85,B 0,C 180,E1 -4423.477,E2 -4423.477} C_VEL
LIN {X 0,Y 532.637,Z 126.545,A -85,B 0,C 180,E1 -4424.78,E2 -4424.78} C_VEL
LIN {X 0,Y 531.224,Z 116.214,A -85,B 0,C 180,E1 -4424.969,E2 -4424.969} C_VEL
LIN {X 0,Y 531.635,Z 94.111,A -85,B 0,C 180,E1 -4428.107,E2 -4428.107} C_VEL
LIN {X 0,Y 531.973,Z 73.33,A -85,B 0,C 180,E1 -4431.1,E2 -4431.1} C_VEL
LIN {X 0,Y 532.39,Z 53.892,A -85,B 0,C 180,E1 -4433.949,E2 -4433.949} C_VEL
LIN {X 0,Y 531.039,Z 46.338,A -85,B 0,C 180,E1 -4435.16,E2 -4435.16} C_VEL
LIN {X 0,Y 531.016,Z 46.338,A -85,B 0,C 180,E1 -4437.595,E2 -4437.595} C_VEL
LIN {X 0,Y 530.974,Z 46.346,A -85,B 0,C 180,E1 -4440.645,E2 -4440.645} C_VEL
LIN {X 0,Y 530.961,Z 46.347,A -85,B 0,C 180,E1 -4443.774,E2 -4443.774} C_VEL
LIN {X 0,Y 530.969,Z 46.343,A -85,B 0,C 180,E1 -4446.557,E2 -4446.557} C_VEL
LIN {X 0,Y 530.978,Z 46.348,A -85,B 0,C 180,E1 -4449.853,E2 -4449.853} C_VEL
LIN {X 0,Y 530.976,Z 46.341,A -85,B 0,C 180,E1 -4452.456,E2 -4452.456} C_VEL
LIN {X 0,Y 530.976,Z 46.343,A -85,B 0,C 180,E1 -4455.622,E2 -4455.622} C_VEL
LIN {X 0,Y 531.005,Z 46.336,A -85,B 0,C 180,E1 -4458.565,E2 -4458.565} C_VEL
LIN {X 0,Y 530.967,Z 46.349,A -85,B 0,C 180,E1 -4461.346,E2 -4461.346} C_VEL
LIN {X 0,Y 530.981,Z 46.34,A -85,B 0,C 180,E1 -4464.382,E2 -4464.382} C_VEL
LIN {X 0,Y 530.969,Z 46.349,A -85,B 0,C 180,E1 -4467.133,E2 -4467.133} C_VEL
LIN {X 0,Y 530.968,Z 46.34,A -85,B 0,C 180,E1 -4469.803,E2 -4469.803} C_VEL
LIN {X 0,Y 531.014,Z 46.338,A -85,B 0,C 180,E1 -4472.467,E2 -4472.467} C_VEL
LIN {X 0,Y 531.004,Z 46.343,A -85,B 0,C 180,E1 -4474.942,E2 -4474.942} C_VEL
LIN {X 0,Y 530.969,Z 46.341,A -85,B 0,C 180,E1 -4478.247,E2 -4478.247} C_VEL
LIN {X 0,Y 530.994,Z 46.343,A -85,B 0,C 180,E1 -4480.677,E2 -4480.677} C_VEL
LIN {X 0,Y 530.984,Z 46.339,A -85,B 0,C 180,E1 -4483.071,E2 -4483.071} C_VEL
LIN {X 0,Y 531.017,Z 46.335,A -85,B 0,C 180,E1 -4485.436,E2 -4485.436} C_VEL
LIN {X 0,Y 531.035,Z 46.337,A -85,B 0,C 180,E1 -4488.55,E2 -4488.55} C_VEL
LIN {X 0,Y 531.054,Z 46.332,A -85,B 0,C 180,E1 -4491.63,E2 -4491.63} C_VEL
LIN {X 0,Y 531.118,Z 46.323,A -85,B 0,C 180,E1 -4494.685,E2 -4494.685} C_VEL
LIN {X 0,Y 531.136,Z 46.325,A -85,B 0,C 180,E1 -4497.725,E2 -4497.725} C_VEL
LIN {X 0,Y 531.15,Z 46.318,A -85,B 0,C 180,E1 -4500.758,E2 -4500.758} C_VEL
LIN {X 0,Y 531.102,Z 46.323,A -85,B 0,C 180,E1 -4503.034,E2 -4503.034} C_VEL
LIN {X 0,Y 531.071,Z 46.329,A -85,B 0,C 180,E1 -4506.077,E2 -4506.077} C_VEL
LIN {X 0,Y 531.02,Z 46.337,A -85,B 0,C 180,E1 -4509.139,E2 -4509.139} C_VEL
LIN {X 0,Y 531.038,Z 46.331,A -85,B 0,C 180,E1 -4512.225,E2 -4512.225} C_VEL
LIN {X 0,Y 530.994,Z 46.343,A -85,B 0,C 180,E1 -4515.35,E2 -4515.35} C_VEL
LIN {X 0,Y 530.983,Z 46.34,A -85,B 0,C 180,E1 -4518.522,E2 -4518.522} C_VEL
LIN {X 0,Y 530.997,Z 46.342,A -85,B 0,C 180,E1 -4520.938,E2 -4520.938} C_VEL
LIN {X 0,Y 530.968,Z 46.343,A -85,B 0,C 180,E1 -4524.225,E2 -4524.225} C_VEL
LIN {X 0,Y 530.985,Z 46.346,A -85,B 0,C 180,E1 -4526.745,E2 -4526.745} C_VEL
LIN {X 0,Y 530.979,Z 46.338,A -85,B 0,C 180,E1 -4529.323,E2 -4529.323} C_VEL
LIN {X 0,Y 530.964,Z 46.346,A -85,B 0,C 180,E1 -4532.101,E2 -4532.101} C_VEL
LIN {X 0,Y 530.963,Z 46.342,A -85,B 0,C 180,E1 -4534.851,E2 -4534.851} C_VEL
LIN {X 0,Y 530.963,Z 46.343,A -85,B 0,C 180,E1 -4537.508,E2 -4537.508} C_VEL
LIN {X 0,Y 530.951,Z 46.344,A -85,B 0,C 180,E1 -4540.436,E2 -4540.436} C_VEL
LIN {X 0,Y 530.927,Z 46.351,A -85,B 0,C 180,E1 -4543.558,E2 -4543.558} C_VEL
LIN {X 0,Y 530.263,Z 46.433,A -85,B 0,C 180,E1 -4544.191,E2 -4544.191} C_VEL
LIN {X 0,Y 527.422,Z 46.784,A -85,B 0,C 180,E1 -4545.22,E2 -4545.22} C_VEL
LIN {X 0,Y 525.016,Z 47.09,A -85,B 0,C 180,E1 -4546.049,E2 -4546.049} C_VEL
LIN {X 0,Y 523.975,Z 47.215,A -85,B 0,C 180,E1 -4546.689,E2 -4546.689} C_VEL
LIN {X 0,Y 523.886,Z 47.226,A -85,B 0,C 180,E1 -4546.905,E2 -4546.905} C_VEL
LIN {X 0,Y 523.913,Z 47.226,A -85,B 0,C 180,E1 -4549.918,E2 -4549.918} C_VEL
LIN {X 0,Y 523.884,Z 47.227,A -85,B 0,C 180,E1 -4552.866,E2 -4552.866} C_VEL
LIN {X 0,Y 523.919,Z 47.228,A -85,B 0,C 180,E1 -4555.709,E2 -4555.709} C_VEL
LIN {X 0,Y 523.977,Z 47.272,A -85,B 0,C 180,E1 -4557.603,E2 -4557.603} C_VEL
LIN {X 0,Y 524.512,Z 53.056,A -85,B 0,C 180,E1 -4558.817,E2 -4558.817} C_VEL
LIN {X 0,Y 524.293,Z 63.459,A -85,B 0,C 180,E1 -4560.914,E2 -4560.914} C_VEL
LIN {X 0,Y 526.044,Z 71.965,A -85,B 0,C 180,E1 -4561.086,E2 -4561.086} C_VEL
LIN {X 0,Y 525.587,Z 169.6,A -85,B 0,C 180,E1 -4562.447,E2 -4562.447} C_VEL
LIN {X 0,Y 525.42,Z 183.218,A -85,B 0,C 180,E1 -4562.801,E2 -4562.801} C_VEL
LIN {X 0,Y 525.246,Z 195.15,A -85,B 0,C 180,E1 -4563.262,E2 -4563.262} C_VEL
LIN {X 0,Y 524.992,Z 206.48,A -85,B 0,C 180,E1 -4563.846,E2 -4563.846} C_VEL
LIN {X 0,Y 524.65,Z 218.034,A -85,B 0,C 180,E1 -4564.618,E2 -4564.618} C_VEL
LIN {X 0,Y 524.437,Z 228.031,A -85,B 0,C 180,E1 -4565.454,E2 -4565.454} C_VEL
LIN {X 0,Y 524.146,Z 238.089,A -85,B 0,C 180,E1 -4566.491,E2 -4566.491} C_VEL
LIN {X 0,Y 523.952,Z 245.887,A -85,B 0,C 180,E1 -4567.484,E2 -4567.484} C_VEL
LIN {X 0,Y 523.715,Z 253.961,A -85,B 0,C 180,E1 -4568.757,E2 -4568.757} C_VEL
LIN {X 0,Y 523.648,Z 260.029,A -85,B 0,C 180,E1 -4569.967,E2 -4569.967} C_VEL
LIN {X 0,Y 523.489,Z 264.87,A -85,B 0,C 180,E1 -4571.204,E2 -4571.204} C_VEL
LIN {X 0,Y 523.419,Z 268.434,A -85,B 0,C 180,E1 -4572.427,E2 -4572.427} C_VEL
LIN {X 0,Y 523.321,Z 270.864,A -85,B 0,C 180,E1 -4573.619,E2 -4573.619} C_VEL
LIN {X 0,Y 523.323,Z 271.917,A -85,B 0,C 180,E1 -4574.42,E2 -4574.42} C_VEL
LIN {X 0,Y 523.342,Z 272.561,A -85,B 0,C 180,E1 -4575.218,E2 -4575.218} C_VEL
LIN {X 0,Y 523.351,Z 272.804,A -85,B 0,C 180,E1 -4576.012,E2 -4576.012} C_VEL
LIN {X 0,Y 523.335,Z 272.598,A -85,B 0,C 180,E1 -4576.803,E2 -4576.803} C_VEL
LIN {X 0,Y 523.374,Z 271.98,A -85,B 0,C 180,E1 -4577.593,E2 -4577.593} C_VEL
LIN {X 0,Y 523.423,Z 270.666,A -85,B 0,C 180,E1 -4578.574,E2 -4578.574} C_VEL
LIN {X 0,Y 523.465,Z 267.653,A -85,B 0,C 180,E1 -4579.949,E2 -4579.949} C_VEL
LIN {X 0,Y 523.503,Z 264.002,A -85,B 0,C 180,E1 -4581.119,E2 -4581.119} C_VEL
LIN {X 0,Y 523.601,Z 259.238,A -85,B 0,C 180,E1 -4582.287,E2 -4582.287} C_VEL
LIN {X 0,Y 523.76,Z 253.123,A -85,B 0,C 180,E1 -4583.47,E2 -4583.47} C_VEL
LIN {X 0,Y 523.898,Z 245.793,A -85,B 0,C 180,E1 -4584.612,E2 -4584.612} C_VEL
LIN {X 0,Y 524.131,Z 238.197,A -85,B 0,C 180,E1 -4585.578,E2 -4585.578} C_VEL
LIN {X 0,Y 524.41,Z 228.978,A -85,B 0,C 180,E1 -4586.543,E2 -4586.543} C_VEL
LIN {X 0,Y 524.63,Z 218.784,A -85,B 0,C 180,E1 -4587.409,E2 -4587.409} C_VEL
LIN {X 0,Y 524.982,Z 207.445,A -85,B 0,C 180,E1 -4588.178,E2 -4588.178} C_VEL
LIN {X 0,Y 525.188,Z 195.678,A -85,B 0,C 180,E1 -4588.802,E2 -4588.802} C_VEL
LIN {X 0,Y 525.321,Z 182.688,A -85,B 0,C 180,E1 -4589.306,E2 -4589.306} C_VEL
LIN {X 0,Y 525.584,Z 169.6,A -85,B 0,C 180,E1 -4589.641,E2 -4589.641} C_VEL
LIN {X 0,Y 525.865,Z 71.056,A -85,B 0,C 180,E1 -4591.02,E2 -4591.02} C_VEL
LIN {X 0,Y 524.196,Z 63.094,A -85,B 0,C 180,E1 -4591.201,E2 -4591.201} C_VEL
LIN {X 0,Y 524.513,Z 51.99,A -85,B 0,C 180,E1 -4593.457,E2 -4593.457} C_VEL
LIN {X 0,Y 523.984,Z 47.219,A -85,B 0,C 180,E1 -4594.472,E2 -4594.472} C_VEL
LIN {X 0,Y 524.04,Z 47.211,A -85,B 0,C 180,E1 -4596.933,E2 -4596.933} C_VEL
LIN {X 0,Y 523.995,Z 47.21,A -85,B 0,C 180,E1 -4599.262,E2 -4599.262} C_VEL
LIN {X 0,Y 524.006,Z 47.208,A -85,B 0,C 180,E1 -4601.738,E2 -4601.738} C_VEL
LIN {X 0,Y 524,Z 47.21,A -85,B 0,C 180,E1 -4605.052,E2 -4605.052} C_VEL
LIN {X 0,Y 523.954,Z 47.218,A -85,B 0,C 180,E1 -4607.97,E2 -4607.97} C_VEL
LIN {X 0,Y 523.978,Z 47.217,A -85,B 0,C 180,E1 -4610.41,E2 -4610.41} C_VEL
LIN {X 0,Y 523.916,Z 47.219,A -85,B 0,C 180,E1 -4612.894,E2 -4612.894} C_VEL
LIN {X 0,Y 523.99,Z 47.219,A -85,B 0,C 180,E1 -4616.02,E2 -4616.02} C_VEL
LIN {X 0,Y 523.936,Z 47.216,A -85,B 0,C 180,E1 -4618.875,E2 -4618.875} C_VEL
LIN {X 0,Y 523.926,Z 47.222,A -85,B 0,C 180,E1 -4621.544,E2 -4621.544} C_VEL
LIN {X 0,Y 523.947,Z 47.217,A -85,B 0,C 180,E1 -4624.289,E2 -4624.289} C_VEL
LIN {X 0,Y 523.915,Z 47.221,A -85,B 0,C 180,E1 -4627.132,E2 -4627.132} C_VEL
LIN {X 0,Y 523.942,Z 47.217,A -85,B 0,C 180,E1 -4630.13,E2 -4630.13} C_VEL
LIN {X 0,Y 523.939,Z 47.216,A -85,B 0,C 180,E1 -4632.459,E2 -4632.459} C_VEL
LIN {X 0,Y 523.946,Z 47.223,A -85,B 0,C 180,E1 -4635.31,E2 -4635.31} C_VEL
LIN {X 0,Y 523.96,Z 47.215,A -85,B 0,C 180,E1 -4638.69,E2 -4638.69} C_VEL
LIN {X 0,Y 523.923,Z 47.226,A -85,B 0,C 180,E1 -4641.08,E2 -4641.08} C_VEL
LIN {X 0,Y 523.904,Z 47.221,A -85,B 0,C 180,E1 -4643.825,E2 -4643.825} C_VEL
LIN {X 0,Y 523.945,Z 47.219,A -85,B 0,C 180,E1 -4646.635,E2 -4646.635} C_VEL
LIN {X 0,Y 523.959,Z 47.216,A -85,B 0,C 180,E1 -4649.355,E2 -4649.355} C_VEL
LIN {X 0,Y 523.98,Z 47.213,A -85,B 0,C 180,E1 -4652.281,E2 -4652.281} C_VEL
LIN {X 0,Y 523.957,Z 47.221,A -85,B 0,C 180,E1 -4654.581,E2 -4654.581} C_VEL
LIN {X 0,Y 523.919,Z 47.221,A -85,B 0,C 180,E1 -4657.106,E2 -4657.106} C_VEL
LIN {X 0,Y 523.982,Z 47.212,A -85,B 0,C 180,E1 -4659.866,E2 -4659.866} C_VEL
LIN {X 0,Y 523.97,Z 47.215,A -85,B 0,C 180,E1 -4662.837,E2 -4662.837} C_VEL
LIN {X 0,Y 523.98,Z 47.211,A -85,B 0,C 180,E1 -4665.236,E2 -4665.236} C_VEL
LIN {X 0,Y 524.016,Z 47.212,A -85,B 0,C 180,E1 -4668.394,E2 -4668.394} C_VEL
LIN {X 0,Y 524.003,Z 47.21,A -85,B 0,C 180,E1 -4671.516,E2 -4671.516} C_VEL
LIN {X 0,Y 524.082,Z 47.199,A -85,B 0,C 180,E1 -4674.613,E2 -4674.613} C_VEL
LIN {X 0,Y 524.112,Z 47.201,A -85,B 0,C 180,E1 -4677.694,E2 -4677.694} C_VEL
LIN {X 0,Y 524.124,Z 47.193,A -85,B 0,C 180,E1 -4680.768,E2 -4680.768} C_VEL
LIN {X 0,Y 524.071,Z 47.201,A -85,B 0,C 180,E1 -4683.075,E2 -4683.075} C_VEL
LIN {X 0,Y 524.037,Z 47.205,A -85,B 0,C 180,E1 -4686.159,E2 -4686.159} C_VEL
LIN {X 0,Y 523.994,Z 47.215,A -85,B 0,C 180,E1 -4689.262,E2 -4689.262} C_VEL
LIN {X 0,Y 524.005,Z 47.211,A -85,B 0,C 180,E1 -4691.739,E2 -4691.739} C_VEL
LIN {X 0,Y 523.995,Z 47.215,A -85,B 0,C 180,E1 -4695.052,E2 -4695.052} C_VEL
LIN {X 0,Y 523.949,Z 47.215,A -85,B 0,C 180,E1 -4697.969,E2 -4697.969} C_VEL
LIN {X 0,Y 523.974,Z 47.213,A -85,B 0,C 180,E1 -4700.41,E2 -4700.41} C_VEL
LIN {X 0,Y 523.912,Z 47.227,A -85,B 0,C 180,E1 -4702.893,E2 -4702.893} C_VEL
LIN {X 0,Y 523.937,Z 47.218,A -85,B 0,C 180,E1 -4705.419,E2 -4705.419} C_VEL
LIN {X 0,Y 523.955,Z 47.214,A -85,B 0,C 180,E1 -4708,E2 -4708} C_VEL
LIN {X 0,Y 523.946,Z 47.222,A -85,B 0,C 180,E1 -4710.855,E2 -4710.855} C_VEL
LIN {X 0,Y 523.961,Z 47.213,A -85,B 0,C 180,E1 -4713.734,E2 -4713.734} C_VEL
LIN {X 0,Y 523.905,Z 47.227,A -85,B 0,C 180,E1 -4716.401,E2 -4716.401} C_VEL
LIN {X 0,Y 523.922,Z 47.219,A -85,B 0,C 180,E1 -4719.085,E2 -4719.085} C_VEL
LIN {X 0,Y 523.953,Z 47.22,A -85,B 0,C 180,E1 -4722.119,E2 -4722.119} C_VEL
LIN {X 0,Y 523.944,Z 47.215,A -85,B 0,C 180,E1 -4725.31,E2 -4725.31} C_VEL
LIN {X 0,Y 523.958,Z 47.215,A -85,B 0,C 180,E1 -4728.69,E2 -4728.69} C_VEL
LIN {X 0,Y 523.918,Z 47.219,A -85,B 0,C 180,E1 -4731.081,E2 -4731.081} C_VEL
LIN {X 0,Y 523.903,Z 47.228,A -85,B 0,C 180,E1 -4733.825,E2 -4733.825} C_VEL
LIN {X 0,Y 523.944,Z 47.216,A -85,B 0,C 180,E1 -4736.636,E2 -4736.636} C_VEL
LIN {X 0,Y 523.952,Z 47.218,A -85,B 0,C 180,E1 -4739.355,E2 -4739.355} C_VEL
LIN {X 0,Y 523.979,Z 47.216,A -85,B 0,C 180,E1 -4742.281,E2 -4742.281} C_VEL
LIN {X 0,Y 524.01,Z 47.385,A -85,B 0,C 180,E1 -4744.717,E2 -4744.717} C_VEL
LIN {X 0,Y 525.407,Z 54.996,A -85,B 0,C 180,E1 -4745.922,E2 -4745.922} C_VEL
LIN {X 0,Y 525.082,Z 71.729,A -85,B 0,C 180,E1 -4748.403,E2 -4748.403} C_VEL
LIN {X 0,Y 524.768,Z 87.012,A -85,B 0,C 180,E1 -4750.642,E2 -4750.642} C_VEL
LIN {X 0,Y 524.407,Z 105.015,A -85,B 0,C 180,E1 -4753.253,E2 -4753.253} C_VEL
LIN {X 0,Y 524.184,Z 115.988,A -85,B 0,C 180,E1 -4754.832,E2 -4754.832} C_VEL
LIN {X 0,Y 525.866,Z 127.938,A -85,B 0,C 180,E1 -4755.048,E2 -4755.048} C_VEL
LIN {X 0,Y 525.476,Z 224.544,A -85,B 0,C 180,E1 -4756.39,E2 -4756.39} C_VEL
LIN {X 0,Y 525.215,Z 237.92,A -85,B 0,C 180,E1 -4756.728,E2 -4756.728} C_VEL
LIN {X 0,Y 524.982,Z 251.282,A -85,B 0,C 180,E1 -4757.239,E2 -4757.239} C_VEL
LIN {X 0,Y 524.678,Z 262.888,A -85,B 0,C 180,E1 -4757.845,E2 -4757.845} C_VEL
LIN {X 0,Y 524.445,Z 274.148,A -85,B 0,C 180,E1 -4758.599,E2 -4758.599} C_VEL
LIN {X 0,Y 524.175,Z 284.641,A -85,B 0,C 180,E1 -4759.474,E2 -4759.474} C_VEL
LIN {X 0,Y 523.903,Z 293.221,A -85,B 0,C 180,E1 -4760.347,E2 -4760.347} C_VEL
LIN {X 0,Y 523.707,Z 301.143,A -85,B 0,C 180,E1 -4761.316,E2 -4761.316} C_VEL
LIN {X 0,Y 523.558,Z 308.884,A -85,B 0,C 180,E1 -4762.479,E2 -4762.479} C_VEL
LIN {X 0,Y 523.431,Z 316.019,A -85,B 0,C 180,E1 -4763.833,E2 -4763.833} C_VEL
LIN {X 0,Y 523.382,Z 320.768,A -85,B 0,C 180,E1 -4764.992,E2 -4764.992} C_VEL
LIN {X 0,Y 523.443,Z 324.401,A -85,B 0,C 180,E1 -4766.15,E2 -4766.15} C_VEL
LIN {X 0,Y 523.417,Z 326.272,A -85,B 0,C 180,E1 -4766.921,E2 -4766.921} C_VEL
LIN {X 0,Y 523.338,Z 327.672,A -85,B 0,C 180,E1 -4767.691,E2 -4767.691} C_VEL
LIN {X 0,Y 523.279,Z 329.279,A -85,B 0,C 180,E1 -4769.23,E2 -4769.23} C_VEL
LIN {X 0,Y 523.283,Z 329.495,A -85,B 0,C 180,E1 -4770,E2 -4770} C_VEL
LIN {X 0,Y 523.279,Z 329.276,A -85,B 0,C 180,E1 -4770.769,E2 -4770.769} C_VEL
LIN {X 0,Y 523.338,Z 327.663,A -85,B 0,C 180,E1 -4772.309,E2 -4772.309} C_VEL
LIN {X 0,Y 523.416,Z 326.26,A -85,B 0,C 180,E1 -4773.078,E2 -4773.078} C_VEL
LIN {X 0,Y 523.422,Z 323.303,A -85,B 0,C 180,E1 -4774.235,E2 -4774.235} C_VEL
LIN {X 0,Y 523.453,Z 319.302,A -85,B 0,C 180,E1 -4775.393,E2 -4775.393} C_VEL
LIN {X 0,Y 523.486,Z 313.246,A -85,B 0,C 180,E1 -4776.727,E2 -4776.727} C_VEL
LIN {X 0,Y 523.634,Z 306.431,A -85,B 0,C 180,E1 -4777.907,E2 -4777.907} C_VEL
LIN {X 0,Y 523.774,Z 298.097,A -85,B 0,C 180,E1 -4779.071,E2 -4779.071} C_VEL
LIN {X 0,Y 523.976,Z 289.558,A -85,B 0,C 180,E1 -4780.041,E2 -4780.041} C_VEL
LIN {X 0,Y 524.284,Z 279.016,A -85,B 0,C 180,E1 -4781.012,E2 -4781.012} C_VEL
LIN {X 0,Y 524.548,Z 267.398,A -85,B 0,C 180,E1 -4781.871,E2 -4781.871} C_VEL
LIN {X 0,Y 524.886,Z 255.227,A -85,B 0,C 180,E1 -4782.567,E2 -4782.567} C_VEL
LIN {X 0,Y 525.13,Z 242.822,A -85,B 0,C 180,E1 -4783.101,E2 -4783.101} C_VEL
LIN {X 0,Y 525.342,Z 230.083,A -85,B 0,C 180,E1 -4783.49,E2 -4783.49} C_VEL
LIN {X 0,Y 525.556,Z 216.711,A -85,B 0,C 180,E1 -4783.731,E2 -4783.731} C_VEL
LIN {X 0,Y 525.724,Z 126.732,A -85,B 0,C 180,E1 -4784.971,E2 -4784.971} C_VEL
LIN {X 0,Y 524.203,Z 115.804,A -85,B 0,C 180,E1 -4785.176,E2 -4785.176} C_VEL
LIN {X 0,Y 524.676,Z 92.544,A -85,B 0,C 180,E1 -4788.529,E2 -4788.529} C_VEL
LIN {X 0,Y 525.041,Z 72.989,A -85,B 0,C 180,E1 -4791.392,E2 -4791.392} C_VEL
LIN {X 0,Y 525.43,Z 54.992,A -85,B 0,C 180,E1 -4794.076,E2 -4794.076} C_VEL
LIN {X 0,Y 524.001,Z 47.214,A -85,B 0,C 180,E1 -4795.363,E2 -4795.363} C_VEL
LIN {X 0,Y 523.97,Z 47.22,A -85,B 0,C 180,E1 -4797.998,E2 -4797.998} C_VEL
LIN {X 0,Y 523.945,Z 47.22,A -85,B 0,C 180,E1 -4800.854,E2 -4800.854} C_VEL
LIN {X 0,Y 523.933,Z 47.222,A -85,B 0,C 180,E1 -4803.73,E2 -4803.73} C_VEL
LIN {X 0,Y 523.923,Z 47.223,A -85,B 0,C 180,E1 -4806.404,E2 -4806.404} C_VEL
LIN {X 0,Y 523.919,Z 47.22,A -85,B 0,C 180,E1 -4809.084,E2 -4809.084} C_VEL
LIN {X 0,Y 523.95,Z 47.219,A -85,B 0,C 180,E1 -4812.119,E2 -4812.119} C_VEL
LIN {X 0,Y 523.942,Z 47.219,A -85,B 0,C 180,E1 -4815.31,E2 -4815.31} C_VEL
LIN {X 0,Y 523.971,Z 47.213,A -85,B 0,C 180,E1 -4818.687,E2 -4818.687} C_VEL
LIN {X 0,Y 523.924,Z 47.223,A -85,B 0,C 180,E1 -4821.079,E2 -4821.079} C_VEL
LIN {X 0,Y 523.927,Z 47.22,A -85,B 0,C 180,E1 -4823.827,E2 -4823.827} C_VEL
LIN {X 0,Y 523.941,Z 47.217,A -85,B 0,C 180,E1 -4826.636,E2 -4826.636} C_VEL
LIN {X 0,Y 523.954,Z 47.218,A -85,B 0,C 180,E1 -4829.356,E2 -4829.356} C_VEL
LIN {X 0,Y 523.977,Z 47.213,A -85,B 0,C 180,E1 -4832.281,E2 -4832.281} C_VEL
LIN {X 0,Y 523.951,Z 47.219,A -85,B 0,C 180,E1 -4834.581,E2 -4834.581} C_VEL
LIN {X 0,Y 523.915,Z 47.219,A -85,B 0,C 180,E1 -4837.107,E2 -4837.107} C_VEL
LIN {X 0,Y 523.977,Z 47.212,A -85,B 0,C 180,E1 -4839.866,E2 -4839.866} C_VEL
LIN {X 0,Y 523.965,Z 47.216,A -85,B 0,C 180,E1 -4842.837,E2 -4842.837} C_VEL
LIN {X 0,Y 523.975,Z 47.212,A -85,B 0,C 180,E1 -4845.236,E2 -4845.236} C_VEL
LIN {X 0,Y 524.01,Z 47.214,A -85,B 0,C 180,E1 -4848.394,E2 -4848.394} C_VEL
